LIN {X 0,Y 573.325,Z 84.689,A -85,B 0,C 180,E1 -2340.7,E2 -2340.7} C_VEL
LIN {X 0,Y 573.297,Z 84.693,A -85,B 0,C 180,E1 -2342.808,E2 -2342.808} C_VEL
LIN {X 0,Y 573.291,Z 84.697,A -85,B 0,C 180,E1 -2345.626,E2 -2345.626} C_VEL
LIN {X 0,Y 573.254,Z 84.699,A -85,B 0,C 180,E1 -2348.457,E2 -2348.457} C_VEL
LIN {X 0,Y 573.274,Z 84.699,A -85,B 0,C 180,E1 -2351.309,E2 -2351.309} C_VEL
LIN {X 0,Y 573.262,Z 84.697,A -85,B 0,C 180,E1 -2354.414,E2 -2354.414} C_VEL
LIN {X 0,Y 573.247,Z 84.702,A -85,B 0,C 180,E1 -2357.109,E2 -2357.109} C_VEL
LIN {X 0,Y 573.233,Z 84.701,A -85,B 0,C 180,E1 -2360.074,E2 -2360.074} C_VEL
LIN {X 0,Y 573.225,Z 84.702,A -85,B 0,C 180,E1 -2362.335,E2 -2362.335} C_VEL
LIN {X 0,Y 573.21,Z 84.704,A -85,B 0,C 180,E1 -2364.357,E2 -2364.357} C_VEL
LIN {X 0,Y 572.573,Z 84.79,A -85,B 0,C 180,E1 -2364.944,E2 -2364.944} C_VEL
LIN {X 0,Y 569.748,Z 85.144,A -85,B 0,C 180,E1 -2365.895,E2 -2365.895} C_VEL
LIN {X 0,Y 567.335,Z 85.445,A -85,B 0,C 180,E1 -2366.661,E2 -2366.661} C_VEL
LIN {X 0,Y 566.283,Z 85.573,A -85,B 0,C 180,E1 -2367.252,E2 -2367.252} C_VEL
LIN {X 0,Y 566.19,Z 85.582,A -85,B 0,C 180,E1 -2367.453,E2 -2367.453} C_VEL
LIN {X 0,Y 566.185,Z 85.576,A -85,B 0,C 180,E1 -2369.766,E2 -2369.766} C_VEL
LIN {X 0,Y 566.19,Z 85.581,A -85,B 0,C 180,E1 -2372.426,E2 -2372.426} C_VEL
LIN {X 0,Y 566.167,Z 85.588,A -85,B 0,C 180,E1 -2374.986,E2 -2374.986} C_VEL
LIN {X 0,Y 566.179,Z 85.579,A -85,B 0,C 180,E1 -2377.458,E2 -2377.458} C_VEL
LIN {X 0,Y 566.188,Z 85.583,A -85,B 0,C 180,E1 -2380.196,E2 -2380.196} C_VEL
LIN {X 0,Y 566.182,Z 85.582,A -85,B 0,C 180,E1 -2383.051,E2 -2383.051} C_VEL
LIN {X 0,Y 566.171,Z 85.585,A -85,B 0,C 180,E1 -2386.046,E2 -2386.046} C_VEL
LIN {X 0,Y 566.179,Z 85.583,A -85,B 0,C 180,E1 -2389.212,E2 -2389.212} C_VEL
LIN {X 0,Y 566.178,Z 85.589,A -85,B 0,C 180,E1 -2392.087,E2 -2392.087} C_VEL
LIN {X 0,Y 566.191,Z 85.725,A -85,B 0,C 180,E1 -2392.454,E2 -2392.454} C_VEL
LIN {X 0,Y 566.912,Z 90.584,A -85,B 0,C 180,E1 -2393.261,E2 -2393.261} C_VEL
LIN {X 0,Y 566.616,Z 108.38,A -85,B 0,C 180,E1 -2396.071,E2 -2396.071} C_VEL
LIN {X 0,Y 566.568,Z 114.772,A -85,B 0,C 180,E1 -2397.07,E2 -2397.07} C_VEL
LIN {X 0,Y 567.79,Z 122.54,A -85,B 0,C 180,E1 -2397.221,E2 -2397.221} C_VEL
LIN {X 0,Y 567.456,Z 251.252,A -85,B 0,C 180,E1 -2398.889,E2 -2398.889} C_VEL
LIN {X 0,Y 567.291,Z 265.503,A -85,B 0,C 180,E1 -2399.215,E2 -2399.215} C_VEL
LIN {X 0,Y 567.168,Z 279.065,A -85,B 0,C 180,E1 -2399.671,E2 -2399.671} C_VEL
LIN {X 0,Y 566.965,Z 292.537,A -85,B 0,C 180,E1 -2400.274,E2 -2400.274} C_VEL
LIN {X 0,Y 566.763,Z 304.844,A -85,B 0,C 180,E1 -2400.976,E2 -2400.976} C_VEL
LIN {X 0,Y 566.577,Z 316.448,A -85,B 0,C 180,E1 -2401.791,E2 -2401.791} C_VEL
LIN {X 0,Y 566.434,Z 326.814,A -85,B 0,C 180,E1 -2402.672,E2 -2402.672} C_VEL
LIN {X 0,Y 566.277,Z 336.543,A -85,B 0,C 180,E1 -2403.66,E2 -2403.66} C_VEL
LIN {X 0,Y 566.136,Z 346.301,A -85,B 0,C 180,E1 -2404.857,E2 -2404.857} C_VEL
LIN {X 0,Y 566.039,Z 353.975,A -85,B 0,C 180,E1 -2406.006,E2 -2406.006} C_VEL
LIN {X 0,Y 565.976,Z 359.753,A -85,B 0,C 180,E1 -2407.05,E2 -2407.05} C_VEL
LIN {X 0,Y 565.952,Z 365.875,A -85,B 0,C 180,E1 -2408.421,E2 -2408.421} C_VEL
LIN {X 0,Y 565.893,Z 370.084,A -85,B 0,C 180,E1 -2409.65,E2 -2409.65} C_VEL
LIN {X 0,Y 565.895,Z 372.821,A -85,B 0,C 180,E1 -2410.698,E2 -2410.698} C_VEL
LIN {X 0,Y 565.829,Z 375.002,A -85,B 0,C 180,E1 -2411.909,E2 -2411.909} C_VEL
LIN {X 0,Y 565.849,Z 376.362,A -85,B 0,C 180,E1 -2413.4,E2 -2413.4} C_VEL
LIN {X 0,Y 565.844,Z 376.254,A -85,B 0,C 180,E1 -2414.88,E2 -2414.88} C_VEL
LIN {X 0,Y 565.917,Z 375.67,A -85,B 0,C 180,E1 -2415.618,E2 -2415.618} C_VEL
LIN {X 0,Y 565.859,Z 373.452,A -85,B 0,C 180,E1 -2417.081,E2 -2417.081} C_VEL
LIN {X 0,Y 565.91,Z 369.79,A -85,B 0,C 180,E1 -2418.538,E2 -2418.538} C_VEL
LIN {X 0,Y 565.919,Z 366.053,A -85,B 0,C 180,E1 -2419.625,E2 -2419.625} C_VEL
LIN {X 0,Y 565.944,Z 361.413,A -85,B 0,C 180,E1 -2420.709,E2 -2420.709} C_VEL
LIN {X 0,Y 566.021,Z 354.686,A -85,B 0,C 180,E1 -2421.969,E2 -2421.969} C_VEL
LIN {X 0,Y 566.131,Z 346.236,A -85,B 0,C 180,E1 -2423.242,E2 -2423.242} C_VEL
LIN {X 0,Y 566.262,Z 337.713,A -85,B 0,C 180,E1 -2424.301,E2 -2424.301} C_VEL
LIN {X 0,Y 566.408,Z 327.309,A -85,B 0,C 180,E1 -2425.373,E2 -2425.373} C_VEL
LIN {X 0,Y 566.578,Z 315.73,A -85,B 0,C 180,E1 -2426.354,E2 -2426.354} C_VEL
LIN {X 0,Y 566.74,Z 304.194,A -85,B 0,C 180,E1 -2427.156,E2 -2427.156} C_VEL
LIN {X 0,Y 566.982,Z 291.521,A -85,B 0,C 180,E1 -2427.868,E2 -2427.868} C_VEL
LIN {X 0,Y 567.18,Z 278.421,A -85,B 0,C 180,E1 -2428.446,E2 -2428.446} C_VEL
LIN {X 0,Y 567.309,Z 264.238,A -85,B 0,C 180,E1 -2428.912,E2 -2428.912} C_VEL
LIN {X 0,Y 567.408,Z 250.022,A -85,B 0,C 180,E1 -2429.223,E2 -2429.223} C_VEL
LIN {X 0,Y 567.634,Z 120.855,A -85,B 0,C 180,E1 -2430.896,E2 -2430.896} C_VEL
LIN {X 0,Y 566.54,Z 114.763,A -85,B 0,C 180,E1 -2431.021,E2 -2431.021} C_VEL
LIN {X 0,Y 566.822,Z 95.22,A -85,B 0,C 180,E1 -2434.087,E2 -2434.087} C_VEL
LIN {X 0,Y 566.763,Z 88.525,A -85,B 0,C 180,E1 -2435.157,E2 -2435.157} C_VEL
LIN {X 0,Y 566.246,Z 85.58,A -85,B 0,C 180,E1 -2435.653,E2 -2435.653} C_VEL
LIN {X 0,Y 566.23,Z 85.582,A -85,B 0,C 180,E1 -2437.846,E2 -2437.846} C_VEL
LIN {X 0,Y 566.226,Z 85.575,A -85,B 0,C 180,E1 -2440.729,E2 -2440.729} C_VEL
LIN {X 0,Y 566.198,Z 85.587,A -85,B 0,C 180,E1 -2443.64,E2 -2443.64} C_VEL
LIN {X 0,Y 566.208,Z 85.575,A -85,B 0,C 180,E1 -2446.587,E2 -2446.587} C_VEL
LIN {X 0,Y 566.181,Z 85.588,A -85,B 0,C 180,E1 -2449.58,E2 -2449.58} C_VEL
LIN {X 0,Y 566.205,Z 85.576,A -85,B 0,C 180,E1 -2452.629,E2 -2452.629} C_VEL
LIN {X 0,Y 566.198,Z 85.58,A -85,B 0,C 180,E1 -2455.748,E2 -2455.748} C_VEL
LIN {X 0,Y 566.208,Z 85.575,A -85,B 0,C 180,E1 -2458.212,E2 -2458.212} C_VEL
LIN {X 0,Y 566.179,Z 85.587,A -85,B 0,C 180,E1 -2461.082,E2 -2461.082} C_VEL
LIN {X 0,Y 566.199,Z 85.578,A -85,B 0,C 180,E1 -2463.739,E2 -2463.739} C_VEL
LIN {X 0,Y 566.195,Z 85.58,A -85,B 0,C 180,E1 -2466.569,E2 -2466.569} C_VEL
LIN {X 0,Y 566.241,Z 85.572,A -85,B 0,C 180,E1 -2469.695,E2 -2469.695} C_VEL
LIN {X 0,Y 566.196,Z 85.577,A -85,B 0,C 180,E1 -2472.087,E2 -2472.087} C_VEL
LIN {X 0,Y 566.191,Z 85.583,A -85,B 0,C 180,E1 -2475.032,E2 -2475.032} C_VEL
LIN {X 0,Y 566.202,Z 85.578,A -85,B 0,C 180,E1 -2478.136,E2 -2478.136} C_VEL
LIN {X 0,Y 566.199,Z 85.584,A -85,B 0,C 180,E1 -2480.73,E2 -2480.73} C_VEL
LIN {X 0,Y 566.202,Z 85.577,A -85,B 0,C 180,E1 -2483.784,E2 -2483.784} C_VEL
LIN {X 0,Y 566.204,Z 85.583,A -85,B 0,C 180,E1 -2486.265,E2 -2486.265} C_VEL
LIN {X 0,Y 566.181,Z 85.58,A -85,B 0,C 180,E1 -2488.923,E2 -2488.923} C_VEL
LIN {X 0,Y 566.204,Z 85.579,A -85,B 0,C 180,E1 -2491.795,E2 -2491.795} C_VEL
LIN {X 0,Y 566.208,Z 85.583,A -85,B 0,C 180,E1 -2494.254,E2 -2494.254} C_VEL
LIN {X 0,Y 566.225,Z 85.575,A -85,B 0,C 180,E1 -2496.703,E2 -2496.703} C_VEL
LIN {X 0,Y 566.206,Z 85.58,A -85,B 0,C 180,E1 -2499.666,E2 -2499.666} C_VEL
LIN {X 0,Y 566.189,Z 85.578,A -85,B 0,C 180,E1 -2502.671,E2 -2502.671} C_VEL
LIN {X 0,Y 566.218,Z 85.581,A -85,B 0,C 180,E1 -2505.629,E2 -2505.629} C_VEL
LIN {X 0,Y 566.26,Z 85.569,A -85,B 0,C 180,E1 -2508.656,E2 -2508.656} C_VEL
LIN {X 0,Y 566.238,Z 85.578,A -85,B 0,C 180,E1 -2511.437,E2 -2511.437} C_VEL
LIN {X 0,Y 566.253,Z 85.57,A -85,B 0,C 180,E1 -2514.304,E2 -2514.304} C_VEL
LIN {X 0,Y 566.269,Z 85.571,A -85,B 0,C 180,E1 -2517.869,E2 -2517.869} C_VEL
LIN {X 0,Y 566.3,Z 85.565,A -85,B 0,C 180,E1 -2520.713,E2 -2520.713} C_VEL
LIN {X 0,Y 566.27,Z 85.571,A -85,B 0,C 180,E1 -2522.848,E2 -2522.848} C_VEL
LIN {X 0,Y 566.253,Z 85.572,A -85,B 0,C 180,E1 -2525.701,E2 -2525.701} C_VEL
LIN {X 0,Y 566.227,Z 85.575,A -85,B 0,C 180,E1 -2528.568,E2 -2528.568} C_VEL
LIN {X 0,Y 566.235,Z 85.575,A -85,B 0,C 180,E1 -2531.456,E2 -2531.456} C_VEL
LIN {X 0,Y 566.228,Z 85.577,A -85,B 0,C 180,E1 -2534.509,E2 -2534.509} C_VEL
LIN {X 0,Y 566.194,Z 85.579,A -85,B 0,C 180,E1 -2537.334,E2 -2537.334} C_VEL
LIN {X 0,Y 566.209,Z 85.579,A -85,B 0,C 180,E1 -2540.339,E2 -2540.339} C_VEL
LIN {X 0,Y 566.185,Z 85.579,A -85,B 0,C 180,E1 -2543.406,E2 -2543.406} C_VEL
LIN {X 0,Y 566.221,Z 85.574,A -85,B 0,C 180,E1 -2545.75,E2 -2545.75} C_VEL
LIN {X 0,Y 566.203,Z 85.581,A -85,B 0,C 180,E1 -2548.205,E2 -2548.205} C_VEL
LIN {X 0,Y 566.187,Z 85.579,A -85,B 0,C 180,E1 -2551.078,E2 -2551.078} C_VEL
LIN {X 0,Y 566.208,Z 85.577,A -85,B 0,C 180,E1 -2553.736,E2 -2553.736} C_VEL
LIN {X 0,Y 566.208,Z 85.579,A -85,B 0,C 180,E1 -2556.571,E2 -2556.571} C_VEL
LIN {X 0,Y 566.213,Z 85.578,A -85,B 0,C 180,E1 -2559.687,E2 -2559.687} C_VEL
LIN {X 0,Y 566.212,Z 85.584,A -85,B 0,C 180,E1 -2562.089,E2 -2562.089} C_VEL
LIN {X 0,Y 566.172,Z 85.58,A -85,B 0,C 180,E1 -2565.037,E2 -2565.037} C_VEL
LIN {X 0,Y 566.211,Z 85.58,A -85,B 0,C 180,E1 -2568.138,E2 -2568.138} C_VEL
LIN {X 0,Y 566.213,Z 85.575,A -85,B 0,C 180,E1 -2570.728,E2 -2570.728} C_VEL
LIN {X 0,Y 566.183,Z 85.586,A -85,B 0,C 180,E1 -2573.79,E2 -2573.79} C_VEL
LIN {X 0,Y 566.211,Z 85.576,A -85,B 0,C 180,E1 -2576.267,E2 -2576.267} C_VEL
LIN {X 0,Y 566.187,Z 85.581,A -85,B 0,C 180,E1 -2578.926,E2 -2578.926} C_VEL
LIN {X 0,Y 566.212,Z 85.58,A -85,B 0,C 180,E1 -2581.859,E2 -2581.859} C_VEL
LIN {X 0,Y 566.208,Z 85.579,A -85,B 0,C 180,E1 -2584.252,E2 -2584.252} C_VEL
LIN {X 0,Y 566.246,Z 85.676,A -85,B 0,C 180,E1 -2585.286,E2 -2585.286} C_VEL
LIN {X 0,Y 567.327,Z 92.177,A -85,B 0,C 180,E1 -2586.222,E2 -2586.222} C_VEL
LIN {X 0,Y 567.075,Z 112.447,A -85,B 0,C 180,E1 -2588.937,E2 -2588.937} C_VEL
LIN {X 0,Y 566.776,Z 135.267,A -85,B 0,C 180,E1 -2591.942,E2 -2591.942} C_VEL
LIN {X 0,Y 566.668,Z 143.53,A -85,B 0,C 180,E1 -2593.019,E2 -2593.019} C_VEL
LIN {X 0,Y 567.795,Z 150.908,A -85,B 0,C 180,E1 -2593.156,E2 -2593.156} C_VEL
LIN {X 0,Y 567.434,Z 281.941,A -85,B 0,C 180,E1 -2594.856,E2 -2594.856} C_VEL
LIN {X 0,Y 567.269,Z 296.626,A -85,B 0,C 180,E1 -2595.203,E2 -2595.203} C_VEL
LIN {X 0,Y 567.1,Z 310.862,A -85,B 0,C 180,E1 -2595.696,E2 -2595.696} C_VEL
LIN {X 0,Y 566.963,Z 323.66,A -85,B 0,C 180,E1 -2596.287,E2 -2596.287} C_VEL
LIN {X 0,Y 566.786,Z 336.117,A -85,B 0,C 180,E1 -2597.013,E2 -2597.013} C_VEL
LIN {X 0,Y 566.577,Z 347.497,A -85,B 0,C 180,E1 -2597.828,E2 -2597.828} C_VEL
LIN {X 0,Y 566.411,Z 358.022,A -85,B 0,C 180,E1 -2598.738,E2 -2598.738} C_VEL
LIN {X 0,Y 566.247,Z 368.343,A -85,B 0,C 180,E1 -2599.814,E2 -2599.814} C_VEL
LIN {X 0,Y 566.152,Z 376.919,A -85,B 0,C 180,E1 -2600.894,E2 -2600.894} C_VEL
LIN {X 0,Y 566.06,Z 385.123,A -85,B 0,C 180,E1 -2602.152,E2 -2602.152} C_VEL
LIN {X 0,Y 565.967,Z 391.807,A -85,B 0,C 180,E1 -2603.423,E2 -2603.423} C_VEL
LIN {X 0,Y 565.928,Z 396.964,A -85,B 0,C 180,E1 -2604.657,E2 -2604.657} C_VEL
LIN {X 0,Y 565.957,Z 400.447,A -85,B 0,C 180,E1 -2605.728,E2 -2605.728} C_VEL
LIN {X 0,Y 565.874,Z 403.834,A -85,B 0,C 180,E1 -2607.153,E2 -2607.153} C_VEL
LIN {X 0,Y 565.841,Z 405.835,A -85,B 0,C 180,E1 -2608.578,E2 -2608.578} C_VEL
LIN {X 0,Y 565.837,Z 406.5,A -85,B 0,C 180,E1 -2610.001,E2 -2610.001} C_VEL
LIN {X 0,Y 565.841,Z 405.834,A -85,B 0,C 180,E1 -2611.424,E2 -2611.424} C_VEL
LIN {X 0,Y 565.874,Z 403.833,A -85,B 0,C 180,E1 -2612.849,E2 -2612.849} C_VEL
LIN {X 0,Y 565.957,Z 400.443,A -85,B 0,C 180,E1 -2614.274,E2 -2614.274} C_VEL
LIN {X 0,Y 565.986,Z 395.564,A -85,B 0,C 180,E1 -2615.702,E2 -2615.702} C_VEL
LIN {X 0,Y 565.998,Z 391.039,A -85,B 0,C 180,E1 -2616.74,E2 -2616.74} C_VEL
LIN {X 0,Y 566.049,Z 384.03,A -85,B 0,C 180,E1 -2618.03,E2 -2618.03} C_VEL
LIN {X 0,Y 566.178,Z 375.549,A -85,B 0,C 180,E1 -2619.287,E2 -2619.287} C_VEL
LIN {X 0,Y 566.295,Z 366.698,A -85,B 0,C 180,E1 -2620.368,E2 -2620.368} C_VEL
LIN {X 0,Y 566.471,Z 355.976,A -85,B 0,C 180,E1 -2621.451,E2 -2621.451} C_VEL
LIN {X 0,Y 566.632,Z 345.123,A -85,B 0,C 180,E1 -2622.355,E2 -2622.355} C_VEL
LIN {X 0,Y 566.801,Z 333.237,A -85,B 0,C 180,E1 -2623.171,E2 -2623.171} C_VEL
LIN {X 0,Y 567.027,Z 320.076,A -85,B 0,C 180,E1 -2623.896,E2 -2623.896} C_VEL
LIN {X 0,Y 567.236,Z 307.029,A -85,B 0,C 180,E1 -2624.453,E2 -2624.453} C_VEL
LIN {X 0,Y 567.329,Z 293.201,A -85,B 0,C 180,E1 -2624.893,E2 -2624.893} C_VEL
LIN {X 0,Y 567.433,Z 279.065,A -85,B 0,C 180,E1 -2625.192,E2 -2625.192} C_VEL
LIN {X 0,Y 567.737,Z 149.617,A -85,B 0,C 180,E1 -2626.863,E2 -2626.863} C_VEL
LIN {X 0,Y 566.67,Z 143.509,A -85,B 0,C 180,E1 -2626.983,E2 -2626.983} C_VEL
LIN {X 0,Y 566.939,Z 122.534,A -85,B 0,C 180,E1 -2629.725,E2 -2629.725} C_VEL
LIN {X 0,Y 567.157,Z 100.948,A -85,B 0,C 180,E1 -2632.591,E2 -2632.591} C_VEL
LIN {X 0,Y 567.257,Z 90.849,A -85,B 0,C 180,E1 -2633.956,E2 -2633.956} C_VEL
LIN {X 0,Y 566.197,Z 85.587,A -85,B 0,C 180,E1 -2634.743,E2 -2634.743} C_VEL
LIN {X 0,Y 566.202,Z 85.578,A -85,B 0,C 180,E1 -2637.341,E2 -2637.341} C_VEL
LIN {X 0,Y 566.205,Z 85.579,A -85,B 0,C 180,E1 -2639.77,E2 -2639.77} C_VEL
LIN {X 0,Y 566.212,Z 85.584,A -85,B 0,C 180,E1 -2642.43,E2 -2642.43} C_VEL
LIN {X 0,Y 566.187,Z 85.58,A -85,B 0,C 180,E1 -2644.989,E2 -2644.989} C_VEL
LIN {X 0,Y 566.203,Z 85.577,A -85,B 0,C 180,E1 -2647.461,E2 -2647.461} C_VEL
LIN {X 0,Y 566.217,Z 85.581,A -85,B 0,C 180,E1 -2650.199,E2 -2650.199} C_VEL
LIN {X 0,Y 566.198,Z 85.577,A -85,B 0,C 180,E1 -2653.056,E2 -2653.056} C_VEL
LIN {X 0,Y 566.205,Z 85.583,A -85,B 0,C 180,E1 -2656.049,E2 -2656.049} C_VEL
LIN {X 0,Y 566.215,Z 85.574,A -85,B 0,C 180,E1 -2659.214,E2 -2659.214} C_VEL
LIN {X 0,Y 566.192,Z 85.587,A -85,B 0,C 180,E1 -2661.636,E2 -2661.636} C_VEL
LIN {X 0,Y 566.161,Z 85.582,A -85,B 0,C 180,E1 -2664.306,E2 -2664.306} C_VEL
LIN {X 0,Y 566.211,Z 85.577,A -85,B 0,C 180,E1 -2666.896,E2 -2666.896} C_VEL
LIN {X 0,Y 566.183,Z 85.587,A -85,B 0,C 180,E1 -2669.406,E2 -2669.406} C_VEL
LIN {X 0,Y 566.2,Z 85.577,A -85,B 0,C 180,E1 -2671.855,E2 -2671.855} C_VEL
LIN {X 0,Y 566.25,Z 85.579,A -85,B 0,C 180,E1 -2675.038,E2 -2675.038} C_VEL
LIN {X 0,Y 566.199,Z 85.577,A -85,B 0,C 180,E1 -2678.136,E2 -2678.136} C_VEL
LIN {X 0,Y 566.243,Z 85.575,A -85,B 0,C 180,E1 -2680.613,E2 -2680.613} C_VEL
LIN {X 0,Y 566.212,Z 85.575,A -85,B 0,C 180,E1 -2683.41,E2 -2683.41} C_VEL
LIN {X 0,Y 566.198,Z 85.582,A -85,B 0,C 180,E1 -2686.357,E2 -2686.357} C_VEL
LIN {X 0,Y 566.246,Z 85.579,A -85,B 0,C 180,E1 -2688.674,E2 -2688.674} C_VEL
LIN {X 0,Y 566.211,Z 85.575,A -85,B 0,C 180,E1 -2691.432,E2 -2691.432} C_VEL
LIN {X 0,Y 566.251,Z 85.578,A -85,B 0,C 180,E1 -2694.299,E2 -2694.299} C_VEL
LIN {X 0,Y 566.285,Z 85.569,A -85,B 0,C 180,E1 -2697.864,E2 -2697.864} C_VEL
LIN {X 0,Y 566.297,Z 85.565,A -85,B 0,C 180,E1 -2700.709,E2 -2700.709} C_VEL
LIN {X 0,Y 566.265,Z 85.569,A -85,B 0,C 180,E1 -2702.843,E2 -2702.843} C_VEL
LIN {X 0,Y 566.258,Z 85.574,A -85,B 0,C 180,E1 -2705.696,E2 -2705.696} C_VEL
LIN {X 0,Y 566.206,Z 85.576,A -85,B 0,C 180,E1 -2708.563,E2 -2708.563} C_VEL
LIN {X 0,Y 566.244,Z 85.577,A -85,B 0,C 180,E1 -2711.451,E2 -2711.451} C_VEL
LIN {X 0,Y 566.218,Z 85.575,A -85,B 0,C 180,E1 -2714.497,E2 -2714.497} C_VEL
LIN {X 0,Y 566.19,Z 85.584,A -85,B 0,C 180,E1 -2717.329,E2 -2717.329} C_VEL
LIN {X 0,Y 566.2,Z 85.576,A -85,B 0,C 180,E1 -2720.334,E2 -2720.334} C_VEL
LIN {X 0,Y 566.161,Z 85.59,A -85,B 0,C 180,E1 -2723.277,E2 -2723.277} C_VEL
LIN {X 0,Y 566.195,Z 85.578,A -85,B 0,C 180,E1 -2725.746,E2 -2725.746} C_VEL
LIN {X 0,Y 566.19,Z 85.582,A -85,B 0,C 180,E1 -2727.453,E2 -2727.453} C_VEL
LIN {X 0,Y 565.501,Z 85.666,A -85,B 0,C 180,E1 -2728.046,E2 -2728.046} C_VEL
LIN {X 0,Y 562.635,Z 86.027,A -85,B 0,C 180,E1 -2729.01,E2 -2729.01} C_VEL
LIN {X 0,Y 560.23,Z 86.321,A -85,B 0,C 180,E1 -2729.786,E2 -2729.786} C_VEL
LIN {X 0,Y 559.204,Z 86.447,A -85,B 0,C 180,E1 -2730.384,E2 -2730.384} C_VEL
LIN {X 0,Y 559.123,Z 86.459,A -85,B 0,C 180,E1 -2730.587,E2 -2730.587} C_VEL
LIN {X 0,Y 559.139,Z 86.463,A -85,B 0,C 180,E1 -2732.712,E2 -2732.712} C_VEL
LIN {X 0,Y 559.114,Z 86.462,A -85,B 0,C 180,E1 -2735.321,E2 -2735.321} C_VEL
LIN {X 0,Y 559.113,Z 86.459,A -85,B 0,C 180,E1 -2738.015,E2 -2738.015} C_VEL
LIN {X 0,Y 559.139,Z 86.462,A -85,B 0,C 180,E1 -2740.809,E2 -2740.809} C_VEL
LIN {X 0,Y 559.126,Z 86.46,A -85,B 0,C 180,E1 -2743.193,E2 -2743.193} C_VEL
LIN {X 0,Y 559.114,Z 86.468,A -85,B 0,C 180,E1 -2746.262,E2 -2746.262} C_VEL
LIN {X 0,Y 559.13,Z 86.462,A -85,B 0,C 180,E1 -2749.184,E2 -2749.184} C_VEL
LIN {X 0,Y 559.176,Z 86.575,A -85,B 0,C 180,E1 -2752.282,E2 -2752.282} C_VEL
LIN {X 0,Y 559.989,Z 92.284,A -85,B 0,C 180,E1 -2753.24,E2 -2753.24} C_VEL
LIN {X 0,Y 559.67,Z 109.35,A -85,B 0,C 180,E1 -2755.967,E2 -2755.967} C_VEL
LIN {X 0,Y 559.617,Z 114.96,A -85,B 0,C 180,E1 -2756.852,E2 -2756.852} C_VEL
LIN {X 0,Y 561,Z 122.414,A -85,B 0,C 180,E1 -2757.007,E2 -2757.007} C_VEL
LIN {X 0,Y 560.611,Z 251.638,A -85,B 0,C 180,E1 -2758.704,E2 -2758.704} C_VEL
LIN {X 0,Y 560.421,Z 265.852,A -85,B 0,C 180,E1 -2759.036,E2 -2759.036} C_VEL
LIN {X 0,Y 560.293,Z 279.873,A -85,B 0,C 180,E1 -2759.52,E2 -2759.52} C_VEL
LIN {X 0,Y 560.063,Z 292.156,A -85,B 0,C 180,E1 -2760.078,E2 -2760.078} C_VEL
LIN {X 0,Y 559.837,Z 304.514,A -85,B 0,C 180,E1 -2760.788,E2 -2760.788} C_VEL
LIN {X 0,Y 559.601,Z 317.408,A -85,B 0,C 180,E1 -2761.712,E2 -2761.712} C_VEL
LIN {X 0,Y 559.402,Z 328.703,A -85,B 0,C 180,E1 -2762.705,E2 -2762.705} C_VEL
LIN {X 0,Y 559.223,Z 338.11,A -85,B 0,C 180,E1 -2763.703,E2 -2763.703} C_VEL
LIN {X 0,Y 559.082,Z 346.929,A -85,B 0,C 180,E1 -2764.825,E2 -2764.825} C_VEL
LIN {X 0,Y 558.973,Z 355.021,A -85,B 0,C 180,E1 -2766.078,E2 -2766.078} C_VEL
LIN {X 0,Y 558.884,Z 362.079,A -85,B 0,C 180,E1 -2767.446,E2 -2767.446} C_VEL
LIN {X 0,Y 558.85,Z 366.88,A -85,B 0,C 180,E1 -2768.61,E2 -2768.61} C_VEL
LIN {X 0,Y 558.821,Z 370.587,A -85,B 0,C 180,E1 -2769.765,E2 -2769.765} C_VEL
LIN {X 0,Y 558.786,Z 373.335,A -85,B 0,C 180,E1 -2770.912,E2 -2770.912} C_VEL
LIN {X 0,Y 558.74,Z 375.645,A -85,B 0,C 180,E1 -2772.429,E2 -2772.429} C_VEL
LIN {X 0,Y 558.741,Z 376.482,A -85,B 0,C 180,E1 -2773.934,E2 -2773.934} C_VEL
LIN {X 0,Y 558.782,Z 375.89,A -85,B 0,C 180,E1 -2775.43,E2 -2775.43} C_VEL
LIN {X 0,Y 558.758,Z 373.862,A -85,B 0,C 180,E1 -2776.914,E2 -2776.914} C_VEL
LIN {X 0,Y 558.82,Z 370.391,A -85,B 0,C 180,E1 -2778.39,E2 -2778.39} C_VEL
LIN {X 0,Y 558.847,Z 365.414,A -85,B 0,C 180,E1 -2779.859,E2 -2779.859} C_VEL
LIN {X 0,Y 558.914,Z 358.797,A -85,B 0,C 180,E1 -2781.32,E2 -2781.32} C_VEL
LIN {X 0,Y 559.023,Z 351.462,A -85,B 0,C 180,E1 -2782.595,E2 -2782.595} C_VEL
LIN {X 0,Y 559.124,Z 343.814,A -85,B 0,C 180,E1 -2783.685,E2 -2783.685} C_VEL
LIN {X 0,Y 559.278,Z 334.677,A -85,B 0,C 180,E1 -2784.772,E2 -2784.772} C_VEL
LIN {X 0,Y 559.427,Z 325.61,A -85,B 0,C 180,E1 -2785.676,E2 -2785.676} C_VEL
LIN {X 0,Y 559.656,Z 313.679,A -85,B 0,C 180,E1 -2786.669,E2 -2786.669} C_VEL
LIN {X 0,Y 559.856,Z 301.71,A -85,B 0,C 180,E1 -2787.481,E2 -2787.481} C_VEL
LIN {X 0,Y 560.137,Z 288.323,A -85,B 0,C 180,E1 -2788.201,E2 -2788.201} C_VEL
LIN {X 0,Y 560.333,Z 275.423,A -85,B 0,C 180,E1 -2788.741,E2 -2788.741} C_VEL
LIN {X 0,Y 560.449,Z 261.6,A -85,B 0,C 180,E1 -2789.168,E2 -2789.168} C_VEL
LIN {X 0,Y 560.556,Z 247.05,A -85,B 0,C 180,E1 -2789.46,E2 -2789.46} C_VEL
LIN {X 0,Y 560.931,Z 122.222,A -85,B 0,C 180,E1 -2791.087,E2 -2791.087} C_VEL
LIN {X 0,Y 559.599,Z 114.957,A -85,B 0,C 180,E1 -2791.236,E2 -2791.236} C_VEL
LIN {X 0,Y 559.912,Z 95.543,A -85,B 0,C 180,E1 -2794.318,E2 -2794.318} C_VEL
LIN {X 0,Y 559.83,Z 89.958,A -85,B 0,C 180,E1 -2795.221,E2 -2795.221} C_VEL
LIN {X 0,Y 559.211,Z 86.457,A -85,B 0,C 180,E1 -2795.815,E2 -2795.815} C_VEL
LIN {X 0,Y 559.179,Z 86.453,A -85,B 0,C 180,E1 -2798.673,E2 -2798.673} C_VEL
LIN {X 0,Y 559.171,Z 86.46,A -85,B 0,C 180,E1 -2801.6,E2 -2801.6} C_VEL
LIN {X 0,Y 559.199,Z 86.448,A -85,B 0,C 180,E1 -2804.611,E2 -2804.611} C_VEL
LIN {X 0,Y 559.176,Z 86.46,A -85,B 0,C 180,E1 -2807.555,E2 -2807.555} C_VEL
LIN {X 0,Y 559.158,Z 86.454,A -85,B 0,C 180,E1 -2810.604,E2 -2810.604} C_VEL
LIN {X 0,Y 559.16,Z 86.458,A -85,B 0,C 180,E1 -2813.715,E2 -2813.715} C_VEL
LIN {X 0,Y 559.171,Z 86.452,A -85,B 0,C 180,E1 -2816.096,E2 -2816.096} C_VEL
LIN {X 0,Y 559.151,Z 86.455,A -85,B 0,C 180,E1 -2818.529,E2 -2818.529} C_VEL
LIN {X 0,Y 559.146,Z 86.463,A -85,B 0,C 180,E1 -2821.281,E2 -2821.281} C_VEL
LIN {X 0,Y 559.155,Z 86.454,A -85,B 0,C 180,E1 -2823.955,E2 -2823.955} C_VEL
LIN {X 0,Y 559.172,Z 86.454,A -85,B 0,C 180,E1 -2826.455,E2 -2826.455} C_VEL
LIN {X 0,Y 559.201,Z 86.448,A -85,B 0,C 180,E1 -2829.862,E2 -2829.862} C_VEL
LIN {X 0,Y 559.141,Z 86.464,A -85,B 0,C 180,E1 -2832.744,E2 -2832.744} C_VEL
LIN {X 0,Y 559.156,Z 86.454,A -85,B 0,C 180,E1 -2835.759,E2 -2835.759} C_VEL
LIN {X 0,Y 559.168,Z 86.457,A -85,B 0,C 180,E1 -2838.947,E2 -2838.947} C_VEL
LIN {X 0,Y 559.152,Z 86.456,A -85,B 0,C 180,E1 -2841.193,E2 -2841.193} C_VEL
LIN {X 0,Y 559.157,Z 86.455,A -85,B 0,C 180,E1 -2843.795,E2 -2843.795} C_VEL
LIN {X 0,Y 559.153,Z 86.463,A -85,B 0,C 180,E1 -2846.429,E2 -2846.429} C_VEL
LIN {X 0,Y 559.145,Z 86.456,A -85,B 0,C 180,E1 -2848.984,E2 -2848.984} C_VEL
LIN {X 0,Y 559.159,Z 86.455,A -85,B 0,C 180,E1 -2851.618,E2 -2851.618} C_VEL
LIN {X 0,Y 559.182,Z 86.456,A -85,B 0,C 180,E1 -2853.907,E2 -2853.907} C_VEL
LIN {X 0,Y 559.16,Z 86.453,A -85,B 0,C 180,E1 -2857.072,E2 -2857.072} C_VEL
LIN {X 0,Y 559.17,Z 86.454,A -85,B 0,C 180,E1 -2859.398,E2 -2859.398} C_VEL
LIN {X 0,Y 559.148,Z 86.457,A -85,B 0,C 180,E1 -2862.446,E2 -2862.446} C_VEL
LIN {X 0,Y 559.178,Z 86.455,A -85,B 0,C 180,E1 -2865.444,E2 -2865.444} C_VEL
LIN {X 0,Y 559.21,Z 86.447,A -85,B 0,C 180,E1 -2868.596,E2 -2868.596} C_VEL
LIN {X 0,Y 559.193,Z 86.454,A -85,B 0,C 180,E1 -2871.328,E2 -2871.328} C_VEL
LIN {X 0,Y 559.221,Z 86.446,A -85,B 0,C 180,E1 -2874.232,E2 -2874.232} C_VEL
LIN {X 0,Y 559.237,Z 86.448,A -85,B 0,C 180,E1 -2877.121,E2 -2877.121} C_VEL
LIN {X 0,Y 559.249,Z 86.443,A -85,B 0,C 180,E1 -2880.002,E2 -2880.002} C_VEL
LIN {X 0,Y 559.236,Z 86.448,A -85,B 0,C 180,E1 -2882.884,E2 -2882.884} C_VEL
LIN {X 0,Y 559.222,Z 86.447,A -85,B 0,C 180,E1 -2885.772,E2 -2885.772} C_VEL
LIN {X 0,Y 559.185,Z 86.454,A -85,B 0,C 180,E1 -2888.676,E2 -2888.676} C_VEL
LIN {X 0,Y 559.198,Z 86.45,A -85,B 0,C 180,E1 -2891.603,E2 -2891.603} C_VEL
LIN {X 0,Y 559.193,Z 86.454,A -85,B 0,C 180,E1 -2894.598,E2 -2894.598} C_VEL
LIN {X 0,Y 559.154,Z 86.455,A -85,B 0,C 180,E1 -2897.559,E2 -2897.559} C_VEL
LIN {X 0,Y 559.167,Z 86.452,A -85,B 0,C 180,E1 -2899.839,E2 -2899.839} C_VEL
LIN {X 0,Y 559.137,Z 86.459,A -85,B 0,C 180,E1 -2902.155,E2 -2902.155} C_VEL
LIN {X 0,Y 559.176,Z 86.453,A -85,B 0,C 180,E1 -2905.189,E2 -2905.189} C_VEL
LIN {X 0,Y 559.191,Z 86.45,A -85,B 0,C 180,E1 -2907.713,E2 -2907.713} C_VEL
LIN {X 0,Y 559.15,Z 86.46,A -85,B 0,C 180,E1 -2910.185,E2 -2910.185} C_VEL
LIN {X 0,Y 559.172,Z 86.456,A -85,B 0,C 180,E1 -2912.716,E2 -2912.716} C_VEL
LIN {X 0,Y 559.142,Z 86.456,A -85,B 0,C 180,E1 -2915.325,E2 -2915.325} C_VEL
LIN {X 0,Y 559.131,Z 86.464,A -85,B 0,C 180,E1 -2918.019,E2 -2918.019} C_VEL
LIN {X 0,Y 559.157,Z 86.454,A -85,B 0,C 180,E1 -2920.814,E2 -2920.814} C_VEL
LIN {X 0,Y 559.147,Z 86.455,A -85,B 0,C 180,E1 -2923.198,E2 -2923.198} C_VEL
LIN {X 0,Y 559.139,Z 86.46,A -85,B 0,C 180,E1 -2926.268,E2 -2926.268} C_VEL
LIN {X 0,Y 559.164,Z 86.453,A -85,B 0,C 180,E1 -2928.95,E2 -2928.95} C_VEL
LIN {X 0,Y 559.174,Z 86.453,A -85,B 0,C 180,E1 -2931.193,E2 -2931.193} C_VEL
LIN {X 0,Y 559.138,Z 86.464,A -85,B 0,C 180,E1 -2933.791,E2 -2933.791} C_VEL
LIN {X 0,Y 559.158,Z 86.454,A -85,B 0,C 180,E1 -2936.426,E2 -2936.426} C_VEL
LIN {X 0,Y 559.151,Z 86.458,A -85,B 0,C 180,E1 -2938.982,E2 -2938.982} C_VEL
LIN {X 0,Y 559.168,Z 86.461,A -85,B 0,C 180,E1 -2941.62,E2 -2941.62} C_VEL
LIN {X 0,Y 559.177,Z 86.457,A -85,B 0,C 180,E1 -2943.904,E2 -2943.904} C_VEL
LIN {X 0,Y 559.219,Z 86.62,A -85,B 0,C 180,E1 -2945.106,E2 -2945.106} C_VEL
LIN {X 0,Y 560.437,Z 93.88,A -85,B 0,C 180,E1 -2946.166,E2 -2946.166} C_VEL
LIN {X 0,Y 560.098,Z 115.132,A -85,B 0,C 180,E1 -2949.048,E2 -2949.048} C_VEL
LIN {X 0,Y 559.808,Z 136.525,A -85,B 0,C 180,E1 -2951.899,E2 -2951.899} C_VEL
LIN {X 0,Y 559.699,Z 143.409,A -85,B 0,C 180,E1 -2952.808,E2 -2952.808} C_VEL
LIN {X 0,Y 560.995,Z 150.933,A -85,B 0,C 180,E1 -2952.949,E2 -2952.949} C_VEL
LIN {X 0,Y 560.593,Z 281.834,A -85,B 0,C 180,E1 -2954.667,E2 -2954.667} C_VEL
LIN {X 0,Y 560.441,Z 296.394,A -85,B 0,C 180,E1 -2955.013,E2 -2955.013} C_VEL
LIN {X 0,Y 560.212,Z 310.822,A -85,B 0,C 180,E1 -2955.516,E2 -2955.516} C_VEL
LIN {X 0,Y 560.057,Z 323.657,A -85,B 0,C 180,E1 -2956.115,E2 -2956.115} C_VEL
LIN {X 0,Y 559.841,Z 336.114,A -85,B 0,C 180,E1 -2956.849,E2 -2956.849} C_VEL
LIN {X 0,Y 559.617,Z 347.494,A -85,B 0,C 180,E1 -2957.674,E2 -2957.674} C_VEL
LIN {X 0,Y 559.388,Z 358.77,A -85,B 0,C 180,E1 -2958.666,E2 -2958.666} C_VEL
LIN {X 0,Y 559.239,Z 368.343,A -85,B 0,C 180,E1 -2959.685,E2 -2959.685} C_VEL
LIN {X 0,Y 559.114,Z 376.918,A -85,B 0,C 180,E1 -2960.779,E2 -2960.779} C_VEL
LIN {X 0,Y 558.98,Z 385.124,A -85,B 0,C 180,E1 -2962.051,E2 -2962.051} C_VEL
LIN {X 0,Y 558.895,Z 392.17,A -85,B 0,C 180,E1 -2963.421,E2 -2963.421} C_VEL
LIN {X 0,Y 558.858,Z 396.964,A -85,B 0,C 180,E1 -2964.589,E2 -2964.589} C_VEL
LIN {X 0,Y 558.866,Z 400.447,A -85,B 0,C 180,E1 -2965.674,E2 -2965.674} C_VEL
LIN {X 0,Y 558.795,Z 403.834,A -85,B 0,C 180,E1 -2967.117,E2 -2967.117} C_VEL
LIN {X 0,Y 558.741,Z 405.835,A -85,B 0,C 180,E1 -2968.56,E2 -2968.56} C_VEL
LIN {X 0,Y 558.738,Z 406.5,A -85,B 0,C 180,E1 -2970.001,E2 -2970.001} C_VEL
LIN {X 0,Y 558.741,Z 405.834,A -85,B 0,C 180,E1 -2971.443,E2 -2971.443} C_VEL
LIN {X 0,Y 558.796,Z 403.833,A -85,B 0,C 180,E1 -2972.885,E2 -2972.885} C_VEL
LIN {X 0,Y 558.866,Z 400.444,A -85,B 0,C 180,E1 -2974.328,E2 -2974.328} C_VEL
LIN {X 0,Y 558.915,Z 395.564,A -85,B 0,C 180,E1 -2975.774,E2 -2975.774} C_VEL
LIN {X 0,Y 558.906,Z 390.859,A -85,B 0,C 180,E1 -2976.861,E2 -2976.861} C_VEL
LIN {X 0,Y 558.988,Z 384.029,A -85,B 0,C 180,E1 -2978.132,E2 -2978.132} C_VEL
LIN {X 0,Y 559.119,Z 375.549,A -85,B 0,C 180,E1 -2979.406,E2 -2979.406} C_VEL
LIN {X 0,Y 559.274,Z 366.698,A -85,B 0,C 180,E1 -2980.5,E2 -2980.5} C_VEL
LIN {X 0,Y 559.458,Z 355.975,A -85,B 0,C 180,E1 -2981.596,E2 -2981.596} C_VEL
LIN {X 0,Y 559.643,Z 345.12,A -85,B 0,C 180,E1 -2982.512,E2 -2982.512} C_VEL
LIN {X 0,Y 559.842,Z 333.234,A -85,B 0,C 180,E1 -2983.338,E2 -2983.338} C_VEL
LIN {X 0,Y 560.109,Z 320.065,A -85,B 0,C 180,E1 -2984.071,E2 -2984.071} C_VEL
LIN {X 0,Y 560.356,Z 307.216,A -85,B 0,C 180,E1 -2984.626,E2 -2984.626} C_VEL
LIN {X 0,Y 560.455,Z 293.854,A -85,B 0,C 180,E1 -2985.061,E2 -2985.061} C_VEL
LIN {X 0,Y 560.589,Z 280.443,A -85,B 0,C 180,E1 -2985.358,E2 -2985.358} C_VEL
LIN {X 0,Y 560.883,Z 150.235,A -85,B 0,C 180,E1 -2987.064,E2 -2987.064} C_VEL
LIN {X 0,Y 559.715,Z 143.373,A -85,B 0,C 180,E1 -2987.193,E2 -2987.193} C_VEL
LIN {X 0,Y 560.017,Z 120.78,A -85,B 0,C 180,E1 -2990.19,E2 -2990.19} C_VEL
LIN {X 0,Y 560.387,Z 97.933,A -85,B 0,C 180,E1 -2993.27,E2 -2993.27} C_VEL
LIN {X 0,Y 560.345,Z 92.235,A -85,B 0,C 180,E1 -2994.056,E2 -2994.056} C_VEL
LIN {X 0,Y 559.165,Z 86.462,A -85,B 0,C 180,E1 -2994.919,E2 -2994.919} C_VEL
LIN {X 0,Y 559.149,Z 86.457,A -85,B 0,C 180,E1 -2997.715,E2 -2997.715} C_VEL
LIN {X 0,Y 559.157,Z 86.461,A -85,B 0,C 180,E1 -3000.184,E2 -3000.184} C_VEL
LIN {X 0,Y 559.162,Z 86.46,A -85,B 0,C 180,E1 -3002.716,E2 -3002.716} C_VEL
LIN {X 0,Y 559.132,Z 86.458,A -85,B 0,C 180,E1 -3005.325,E2 -3005.325} C_VEL
LIN {X 0,Y 559.142,Z 86.462,A -85,B 0,C 180,E1 -3008.018,E2 -3008.018} C_VEL
LIN {X 0,Y 559.166,Z 86.453,A -85,B 0,C 180,E1 -3010.813,E2 -3010.813} C_VEL
LIN {X 0,Y 559.122,Z 86.465,A -85,B 0,C 180,E1 -3013.737,E2 -3013.737} C_VEL
LIN {X 0,Y 559.149,Z 86.459,A -85,B 0,C 180,E1 -3016.266,E2 -3016.266} C_VEL
LIN {X 0,Y 559.167,Z 86.451,A -85,B 0,C 180,E1 -3019.187,E2 -3019.187} C_VEL
LIN {X 0,Y 559.14,Z 86.459,A -85,B 0,C 180,E1 -3021.982,E2 -3021.982} C_VEL
LIN {X 0,Y 559.14,Z 86.457,A -85,B 0,C 180,E1 -3024.787,E2 -3024.787} C_VEL
LIN {X 0,Y 559.165,Z 86.462,A -85,B 0,C 180,E1 -3027.364,E2 -3027.364} C_VEL
LIN {X 0,Y 559.134,Z 86.457,A -85,B 0,C 180,E1 -3030.147,E2 -3030.147} C_VEL
LIN {X 0,Y 559.155,Z 86.462,A -85,B 0,C 180,E1 -3033.177,E2 -3033.177} C_VEL
LIN {X 0,Y 559.166,Z 86.455,A -85,B 0,C 180,E1 -3035.494,E2 -3035.494} C_VEL
LIN {X 0,Y 559.183,Z 86.455,A -85,B 0,C 180,E1 -3038.623,E2 -3038.623} C_VEL
LIN {X 0,Y 559.171,Z 86.461,A -85,B 0,C 180,E1 -3040.925,E2 -3040.925} C_VEL
LIN {X 0,Y 559.166,Z 86.452,A -85,B 0,C 180,E1 -3043.946,E2 -3043.946} C_VEL
LIN {X 0,Y 559.172,Z 86.455,A -85,B 0,C 180,E1 -3046.182,E2 -3046.182} C_VEL
LIN {X 0,Y 559.202,Z 86.45,A -85,B 0,C 180,E1 -3049.132,E2 -3049.132} C_VEL
LIN {X 0,Y 559.199,Z 86.452,A -85,B 0,C 180,E1 -3052.051,E2 -3052.051} C_VEL
LIN {X 0,Y 559.25,Z 86.444,A -85,B 0,C 180,E1 -3054.951,E2 -3054.951} C_VEL
LIN {X 0,Y 559.257,Z 86.444,A -85,B 0,C 180,E1 -3057.837,E2 -3057.837} C_VEL
LIN {X 0,Y 559.269,Z 86.44,A -85,B 0,C 180,E1 -3060.718,E2 -3060.718} C_VEL
LIN {X 0,Y 559.233,Z 86.445,A -85,B 0,C 180,E1 -3062.879,E2 -3062.879} C_VEL
LIN {X 0,Y 559.226,Z 86.451,A -85,B 0,C 180,E1 -3065.768,E2 -3065.768} C_VEL
LIN {X 0,Y 559.17,Z 86.452,A -85,B 0,C 180,E1 -3068.672,E2 -3068.672} C_VEL
LIN {X 0,Y 559.207,Z 86.456,A -85,B 0,C 180,E1 -3071.598,E2 -3071.598} C_VEL
LIN {X 0,Y 559.181,Z 86.451,A -85,B 0,C 180,E1 -3074.585,E2 -3074.585} C_VEL
LIN {X 0,Y 559.134,Z 86.465,A -85,B 0,C 180,E1 -3077.555,E2 -3077.555} C_VEL
LIN {X 0,Y 559.161,Z 86.456,A -85,B 0,C 180,E1 -3079.835,E2 -3079.835} C_VEL
LIN {X 0,Y 559.134,Z 86.457,A -85,B 0,C 180,E1 -3082.15,E2 -3082.15} C_VEL
LIN {X 0,Y 559.135,Z 86.466,A -85,B 0,C 180,E1 -3085.175,E2 -3085.175} C_VEL
LIN {X 0,Y 559.138,Z 86.458,A -85,B 0,C 180,E1 -3087.711,E2 -3087.711} C_VEL
LIN {X 0,Y 559.123,Z 86.459,A -85,B 0,C 180,E1 -3090.587,E2 -3090.587} C_VEL
LIN {X 0,Y 558.46,Z 86.548,A -85,B 0,C 180,E1 -3091.189,E2 -3091.189} C_VEL
LIN {X 0,Y 555.597,Z 86.903,A -85,B 0,C 180,E1 -3092.165,E2 -3092.165} C_VEL
LIN {X 0,Y 553.181,Z 87.205,A -85,B 0,C 180,E1 -3092.95,E2 -3092.95} C_VEL
LIN {X 0,Y 552.154,Z 87.326,A -85,B 0,C 180,E1 -3093.557,E2 -3093.557} C_VEL
LIN {X 0,Y 552.076,Z 87.334,A -85,B 0,C 180,E1 -3093.762,E2 -3093.762} C_VEL
LIN {X 0,Y 552.09,Z 87.342,A -85,B 0,C 180,E1 -3096.744,E2 -3096.744} C_VEL
LIN {X 0,Y 552.109,Z 87.333,A -85,B 0,C 180,E1 -3099.524,E2 -3099.524} C_VEL
LIN {X 0,Y 552.113,Z 87.34,A -85,B 0,C 180,E1 -3102.422,E2 -3102.422} C_VEL
LIN {X 0,Y 552.071,Z 87.337,A -85,B 0,C 180,E1 -3105.559,E2 -3105.559} C_VEL
LIN {X 0,Y 552.085,Z 87.343,A -85,B 0,C 180,E1 -3108.677,E2 -3108.677} C_VEL
LIN {X 0,Y 552.095,Z 87.34,A -85,B 0,C 180,E1 -3111.408,E2 -3111.408} C_VEL
LIN {X 0,Y 552.101,Z 87.448,A -85,B 0,C 180,E1 -3112.107,E2 -3112.107} C_VEL
LIN {X 0,Y 553.083,Z 93.704,A -85,B 0,C 180,E1 -3113.175,E2 -3113.175} C_VEL
LIN {X 0,Y 552.69,Z 112.462,A -85,B 0,C 180,E1 -3116.197,E2 -3116.197} C_VEL
LIN {X 0,Y 552.648,Z 115.275,A -85,B 0,C 180,E1 -3116.643,E2 -3116.643} C_VEL
LIN {X 0,Y 554.227,Z 123.884,A -85,B 0,C 180,E1 -3116.81,E2 -3116.81} C_VEL
LIN {X 0,Y 553.782,Z 252.214,A -85,B 0,C 180,E1 -3118.519,E2 -3118.519} C_VEL
LIN {X 0,Y 553.574,Z 266.818,A -85,B 0,C 180,E1 -3118.871,E2 -3118.871} C_VEL
LIN {X 0,Y 553.397,Z 280.727,A -85,B 0,C 180,E1 -3119.363,E2 -3119.363} C_VEL
LIN {X 0,Y 553.152,Z 293.673,A -85,B 0,C 180,E1 -3119.971,E2 -3119.971} C_VEL
LIN {X 0,Y 552.899,Z 305.913,A -85,B 0,C 180,E1 -3120.699,E2 -3120.699} C_VEL
LIN {X 0,Y 552.655,Z 317.79,A -85,B 0,C 180,E1 -3121.571,E2 -3121.571} C_VEL
LIN {X 0,Y 552.436,Z 328.589,A -85,B 0,C 180,E1 -3122.537,E2 -3122.537} C_VEL
LIN {X 0,Y 552.201,Z 337.988,A -85,B 0,C 180,E1 -3123.547,E2 -3123.547} C_VEL
LIN {X 0,Y 552.04,Z 346.673,A -85,B 0,C 180,E1 -3124.665,E2 -3124.665} C_VEL
LIN {X 0,Y 551.896,Z 354.889,A -85,B 0,C 180,E1 -3125.951,E2 -3125.951} C_VEL
LIN {X 0,Y 551.817,Z 361.084,A -85,B 0,C 180,E1 -3127.141,E2 -3127.141} C_VEL
LIN {X 0,Y 551.77,Z 366.335,A -85,B 0,C 180,E1 -3128.394,E2 -3128.394} C_VEL
LIN {X 0,Y 551.719,Z 371.071,A -85,B 0,C 180,E1 -3129.882,E2 -3129.882} C_VEL
LIN {X 0,Y 551.712,Z 372.909,A -85,B 0,C 180,E1 -3130.657,E2 -3130.657} C_VEL
LIN {X 0,Y 551.648,Z 375.411,A -85,B 0,C 180,E1 -3132.195,E2 -3132.195} C_VEL
LIN {X 0,Y 551.645,Z 376.436,A -85,B 0,C 180,E1 -3133.722,E2 -3133.722} C_VEL
LIN {X 0,Y 551.669,Z 376.032,A -85,B 0,C 180,E1 -3135.238,E2 -3135.238} C_VEL
LIN {X 0,Y 551.671,Z 374.223,A -85,B 0,C 180,E1 -3136.743,E2 -3136.743} C_VEL
LIN {X 0,Y 551.71,Z 370.987,A -85,B 0,C 180,E1 -3138.239,E2 -3138.239} C_VEL
LIN {X 0,Y 551.763,Z 367.539,A -85,B 0,C 180,E1 -3139.356,E2 -3139.356} C_VEL
LIN {X 0,Y 551.804,Z 361.601,A -85,B 0,C 180,E1 -3140.838,E2 -3140.838} C_VEL
LIN {X 0,Y 551.897,Z 354.932,A -85,B 0,C 180,E1 -3142.131,E2 -3142.131} C_VEL
LIN {X 0,Y 552.064,Z 346.701,A -85,B 0,C 180,E1 -3143.42,E2 -3143.42} C_VEL
LIN {X 0,Y 552.222,Z 338.169,A -85,B 0,C 180,E1 -3144.522,E2 -3144.522} C_VEL
LIN {X 0,Y 552.4,Z 327.886,A -85,B 0,C 180,E1 -3145.621,E2 -3145.621} C_VEL
LIN {X 0,Y 552.65,Z 316.426,A -85,B 0,C 180,E1 -3146.627,E2 -3146.627} C_VEL
LIN {X 0,Y 552.875,Z 305.026,A -85,B 0,C 180,E1 -3147.449,E2 -3147.449} C_VEL
LIN {X 0,Y 553.172,Z 292.522,A -85,B 0,C 180,E1 -3148.179,E2 -3148.179} C_VEL
LIN {X 0,Y 553.436,Z 279.632,A -85,B 0,C 180,E1 -3148.771,E2 -3148.771} C_VEL
LIN {X 0,Y 553.594,Z 265.831,A -85,B 0,C 180,E1 -3149.249,E2 -3149.249} C_VEL
LIN {X 0,Y 553.719,Z 251.309,A -85,B 0,C 180,E1 -3149.59,E2 -3149.59} C_VEL
LIN {X 0,Y 554.154,Z 123.051,A -85,B 0,C 180,E1 -3151.293,E2 -3151.293} C_VEL
LIN {X 0,Y 552.646,Z 115.167,A -85,B 0,C 180,E1 -3151.456,E2 -3151.456} C_VEL
LIN {X 0,Y 553.006,Z 95.868,A -85,B 0,C 180,E1 -3154.555,E2 -3154.555} C_VEL
LIN {X 0,Y 552.897,Z 91.396,A -85,B 0,C 180,E1 -3155.287,E2 -3155.287} C_VEL
LIN {X 0,Y 552.164,Z 87.335,A -85,B 0,C 180,E1 -3156.004,E2 -3156.004} C_VEL
LIN {X 0,Y 552.146,Z 87.329,A -85,B 0,C 180,E1 -3158.785,E2 -3158.785} C_VEL
LIN {X 0,Y 552.128,Z 87.34,A -85,B 0,C 180,E1 -3161.75,E2 -3161.75} C_VEL
LIN {X 0,Y 552.168,Z 87.324,A -85,B 0,C 180,E1 -3164.746,E2 -3164.746} C_VEL
LIN {X 0,Y 552.108,Z 87.338,A -85,B 0,C 180,E1 -3167.787,E2 -3167.787} C_VEL
LIN {X 0,Y 552.102,Z 87.334,A -85,B 0,C 180,E1 -3170.101,E2 -3170.101} C_VEL
LIN {X 0,Y 552.122,Z 87.33,A -85,B 0,C 180,E1 -3172.448,E2 -3172.448} C_VEL
LIN {X 0,Y 552.145,Z 87.337,A -85,B 0,C 180,E1 -3175.358,E2 -3175.358} C_VEL
LIN {X 0,Y 552.105,Z 87.332,A -85,B 0,C 180,E1 -3178.097,E2 -3178.097} C_VEL
LIN {X 0,Y 552.088,Z 87.336,A -85,B 0,C 180,E1 -3180.609,E2 -3180.609} C_VEL
LIN {X 0,Y 552.107,Z 87.34,A -85,B 0,C 180,E1 -3183.185,E2 -3183.185} C_VEL
LIN {X 0,Y 552.1,Z 87.333,A -85,B 0,C 180,E1 -3185.841,E2 -3185.841} C_VEL
LIN {X 0,Y 552.115,Z 87.338,A -85,B 0,C 180,E1 -3189.067,E2 -3189.067} C_VEL
LIN {X 0,Y 552.142,Z 87.329,A -85,B 0,C 180,E1 -3191.442,E2 -3191.442} C_VEL
LIN {X 0,Y 552.097,Z 87.339,A -85,B 0,C 180,E1 -3194.537,E2 -3194.537} C_VEL
LIN {X 0,Y 552.101,Z 87.333,A -85,B 0,C 180,E1 -3197.586,E2 -3197.586} C_VEL
LIN {X 0,Y 552.124,Z 87.338,A -85,B 0,C 180,E1 -3200.477,E2 -3200.477} C_VEL
LIN {X 0,Y 552.111,Z 87.332,A -85,B 0,C 180,E1 -3203.314,E2 -3203.314} C_VEL
LIN {X 0,Y 552.117,Z 87.333,A -85,B 0,C 180,E1 -3205.943,E2 -3205.943} C_VEL
LIN {X 0,Y 552.109,Z 87.338,A -85,B 0,C 180,E1 -3208.544,E2 -3208.544} C_VEL
LIN {X 0,Y 552.111,Z 87.332,A -85,B 0,C 180,E1 -3211.438,E2 -3211.438} C_VEL
LIN {X 0,Y 552.141,Z 87.334,A -85,B 0,C 180,E1 -3214.36,E2 -3214.36} C_VEL
LIN {X 0,Y 552.131,Z 87.33,A -85,B 0,C 180,E1 -3216.763,E2 -3216.763} C_VEL
LIN {X 0,Y 552.117,Z 87.339,A -85,B 0,C 180,E1 -3219.902,E2 -3219.902} C_VEL
LIN {X 0,Y 552.142,Z 87.328,A -85,B 0,C 180,E1 -3222.98,E2 -3222.98} C_VEL
LIN {X 0,Y 552.123,Z 87.336,A -85,B 0,C 180,E1 -3226.007,E2 -3226.007} C_VEL
LIN {X 0,Y 552.164,Z 87.326,A -85,B 0,C 180,E1 -3228.996,E2 -3228.996} C_VEL
LIN {X 0,Y 552.154,Z 87.33,A -85,B 0,C 180,E1 -3231.954,E2 -3231.954} C_VEL
LIN {X 0,Y 552.225,Z 87.319,A -85,B 0,C 180,E1 -3234.892,E2 -3234.892} C_VEL
LIN {X 0,Y 552.213,Z 87.322,A -85,B 0,C 180,E1 -3237.814,E2 -3237.814} C_VEL
LIN {X 0,Y 552.239,Z 87.317,A -85,B 0,C 180,E1 -3240.732,E2 -3240.732} C_VEL
LIN {X 0,Y 552.202,Z 87.324,A -85,B 0,C 180,E1 -3242.92,E2 -3242.92} C_VEL
LIN {X 0,Y 552.192,Z 87.322,A -85,B 0,C 180,E1 -3245.846,E2 -3245.846} C_VEL
LIN {X 0,Y 552.156,Z 87.331,A -85,B 0,C 180,E1 -3248.788,E2 -3248.788} C_VEL
LIN {X 0,Y 552.156,Z 87.326,A -85,B 0,C 180,E1 -3251.753,E2 -3251.753} C_VEL
LIN {X 0,Y 552.131,Z 87.336,A -85,B 0,C 180,E1 -3254.75,E2 -3254.75} C_VEL
LIN {X 0,Y 552.106,Z 87.332,A -85,B 0,C 180,E1 -3257.791,E2 -3257.791} C_VEL
LIN {X 0,Y 552.126,Z 87.331,A -85,B 0,C 180,E1 -3260.103,E2 -3260.103} C_VEL
LIN {X 0,Y 552.091,Z 87.34,A -85,B 0,C 180,E1 -3262.453,E2 -3262.453} C_VEL
LIN {X 0,Y 552.153,Z 87.327,A -85,B 0,C 180,E1 -3265.353,E2 -3265.353} C_VEL
LIN {X 0,Y 552.123,Z 87.334,A -85,B 0,C 180,E1 -3268.099,E2 -3268.099} C_VEL
LIN {X 0,Y 552.099,Z 87.339,A -85,B 0,C 180,E1 -3270.611,E2 -3270.611} C_VEL
LIN {X 0,Y 552.12,Z 87.33,A -85,B 0,C 180,E1 -3273.187,E2 -3273.187} C_VEL
LIN {X 0,Y 552.1,Z 87.336,A -85,B 0,C 180,E1 -3275.844,E2 -3275.844} C_VEL
LIN {X 0,Y 552.119,Z 87.33,A -85,B 0,C 180,E1 -3279.063,E2 -3279.063} C_VEL
LIN {X 0,Y 552.131,Z 87.33,A -85,B 0,C 180,E1 -3281.446,E2 -3281.446} C_VEL
LIN {X 0,Y 552.095,Z 87.335,A -85,B 0,C 180,E1 -3284.534,E2 -3284.534} C_VEL
LIN {X 0,Y 552.13,Z 87.334,A -85,B 0,C 180,E1 -3287.586,E2 -3287.586} C_VEL
LIN {X 0,Y 552.128,Z 87.33,A -85,B 0,C 180,E1 -3290.474,E2 -3290.474} C_VEL
LIN {X 0,Y 552.105,Z 87.336,A -85,B 0,C 180,E1 -3293.319,E2 -3293.319} C_VEL
LIN {X 0,Y 552.125,Z 87.334,A -85,B 0,C 180,E1 -3295.94,E2 -3295.94} C_VEL
LIN {X 0,Y 552.119,Z 87.332,A -85,B 0,C 180,E1 -3298.542,E2 -3298.542} C_VEL
LIN {X 0,Y 552.124,Z 87.339,A -85,B 0,C 180,E1 -3301.44,E2 -3301.44} C_VEL
LIN {X 0,Y 552.129,Z 87.334,A -85,B 0,C 180,E1 -3304.357,E2 -3304.357} C_VEL
LIN {X 0,Y 552.175,Z 87.385,A -85,B 0,C 180,E1 -3304.897,E2 -3304.897} C_VEL
LIN {X 0,Y 553.569,Z 95.353,A -85,B 0,C 180,E1 -3306.079,E2 -3306.079} C_VEL
LIN {X 0,Y 553.149,Z 116.389,A -85,B 0,C 180,E1 -3308.967,E2 -3308.967} C_VEL
LIN {X 0,Y 552.807,Z 137.753,A -85,B 0,C 180,E1 -3311.853,E2 -3311.853} C_VEL
LIN {X 0,Y 552.726,Z 143.183,A -85,B 0,C 180,E1 -3312.581,E2 -3312.581} C_VEL
LIN {X 0,Y 554.203,Z 151.689,A -85,B 0,C 180,E1 -3312.746,E2 -3312.746} C_VEL
LIN {X 0,Y 553.752,Z 281.588,A -85,B 0,C 180,E1 -3314.473,E2 -3314.473} C_VEL
LIN {X 0,Y 553.567,Z 295.794,A -85,B 0,C 180,E1 -3314.811,E2 -3314.811} C_VEL
LIN {X 0,Y 553.376,Z 309.471,A -85,B 0,C 180,E1 -3315.287,E2 -3315.287} C_VEL
LIN {X 0,Y 553.127,Z 323.445,A -85,B 0,C 180,E1 -3315.937,E2 -3315.937} C_VEL
LIN {X 0,Y 552.869,Z 335.948,A -85,B 0,C 180,E1 -3316.68,E2 -3316.68} C_VEL
LIN {X 0,Y 552.654,Z 347.377,A -85,B 0,C 180,E1 -3317.516,E2 -3317.516} C_VEL
LIN {X 0,Y 552.407,Z 358.707,A -85,B 0,C 180,E1 -3318.52,E2 -3318.52} C_VEL
LIN {X 0,Y 552.227,Z 368.329,A -85,B 0,C 180,E1 -3319.552,E2 -3319.552} C_VEL
LIN {X 0,Y 552.071,Z 376.917,A -85,B 0,C 180,E1 -3320.66,E2 -3320.66} C_VEL
LIN {X 0,Y 551.902,Z 385.125,A -85,B 0,C 180,E1 -3321.949,E2 -3321.949} C_VEL
LIN {X 0,Y 551.824,Z 390.868,A -85,B 0,C 180,E1 -3323.052,E2 -3323.052} C_VEL
LIN {X 0,Y 551.792,Z 396.964,A -85,B 0,C 180,E1 -3324.52,E2 -3324.52} C_VEL
LIN {X 0,Y 551.76,Z 400.447,A -85,B 0,C 180,E1 -3325.618,E2 -3325.618} C_VEL
LIN {X 0,Y 551.719,Z 403.834,A -85,B 0,C 180,E1 -3327.08,E2 -3327.08} C_VEL
LIN {X 0,Y 551.641,Z 405.836,A -85,B 0,C 180,E1 -3328.541,E2 -3328.541} C_VEL
LIN {X 0,Y 551.639,Z 406.5,A -85,B 0,C 180,E1 -3330.001,E2 -3330.001} C_VEL
LIN {X 0,Y 551.641,Z 405.835,A -85,B 0,C 180,E1 -3331.461,E2 -3331.461} C_VEL
LIN {X 0,Y 551.72,Z 403.834,A -85,B 0,C 180,E1 -3332.922,E2 -3332.922} C_VEL
LIN {X 0,Y 551.76,Z 400.444,A -85,B 0,C 180,E1 -3334.384,E2 -3334.384} C_VEL
LIN {X 0,Y 551.824,Z 395.563,A -85,B 0,C 180,E1 -3335.849,E2 -3335.849} C_VEL
LIN {X 0,Y 551.836,Z 389.049,A -85,B 0,C 180,E1 -3337.318,E2 -3337.318} C_VEL
LIN {X 0,Y 551.964,Z 381.797,A -85,B 0,C 180,E1 -3338.605,E2 -3338.605} C_VEL
LIN {X 0,Y 552.118,Z 372.813,A -85,B 0,C 180,E1 -3339.896,E2 -3339.896} C_VEL
LIN {X 0,Y 552.332,Z 363.342,A -85,B 0,C 180,E1 -3341.004,E2 -3341.004} C_VEL
LIN {X 0,Y 552.485,Z 352.842,A -85,B 0,C 180,E1 -3342.024,E2 -3342.024} C_VEL
LIN {X 0,Y 552.717,Z 341.261,A -85,B 0,C 180,E1 -3342.951,E2 -3342.951} C_VEL
LIN {X 0,Y 553.015,Z 328.415,A -85,B 0,C 180,E1 -3343.786,E2 -3343.786} C_VEL
LIN {X 0,Y 553.25,Z 315.869,A -85,B 0,C 180,E1 -3344.437,E2 -3344.437} C_VEL
LIN {X 0,Y 553.471,Z 302.714,A -85,B 0,C 180,E1 -3344.966,E2 -3344.966} C_VEL
LIN {X 0,Y 553.647,Z 288.526,A -85,B 0,C 180,E1 -3345.381,E2 -3345.381} C_VEL
LIN {X 0,Y 553.739,Z 274.104,A -85,B 0,C 180,E1 -3345.648,E2 -3345.648} C_VEL
LIN {X 0,Y 554.199,Z 151.974,A -85,B 0,C 180,E1 -3347.25,E2 -3347.25} C_VEL
LIN {X 0,Y 552.737,Z 143.123,A -85,B 0,C 180,E1 -3347.423,E2 -3347.423} C_VEL
LIN {X 0,Y 553.051,Z 120.589,A -85,B 0,C 180,E1 -3350.455,E2 -3350.455} C_VEL
LIN {X 0,Y 553.525,Z 97.984,A -85,B 0,C 180,E1 -3353.546,E2 -3353.546} C_VEL
LIN {X 0,Y 553.408,Z 93.486,A -85,B 0,C 180,E1 -3354.178,E2 -3354.178} C_VEL
LIN {X 0,Y 552.124,Z 87.338,A -85,B 0,C 180,E1 -3355.103,E2 -3355.103} C_VEL
LIN {X 0,Y 552.13,Z 87.332,A -85,B 0,C 180,E1 -3357.275,E2 -3357.275} C_VEL
LIN {X 0,Y 552.121,Z 87.336,A -85,B 0,C 180,E1 -3360.05,E2 -3360.05} C_VEL
LIN {X 0,Y 552.12,Z 87.336,A -85,B 0,C 180,E1 -3362.846,E2 -3362.846} C_VEL
LIN {X 0,Y 552.08,Z 87.337,A -85,B 0,C 180,E1 -3365.439,E2 -3365.439} C_VEL
LIN {X 0,Y 552.105,Z 87.337,A -85,B 0,C 180,E1 -3367.885,E2 -3367.885} C_VEL
LIN {X 0,Y 552.119,Z 87.333,A -85,B 0,C 180,E1 -3370.481,E2 -3370.481} C_VEL
LIN {X 0,Y 552.104,Z 87.336,A -85,B 0,C 180,E1 -3373.481,E2 -3373.481} C_VEL
LIN {X 0,Y 552.119,Z 87.332,A -85,B 0,C 180,E1 -3376.576,E2 -3376.576} C_VEL
LIN {X 0,Y 552.119,Z 87.333,A -85,B 0,C 180,E1 -3379.518,E2 -3379.518} C_VEL
LIN {X 0,Y 552.099,Z 87.333,A -85,B 0,C 180,E1 -3382.335,E2 -3382.335} C_VEL
LIN {X 0,Y 552.092,Z 87.337,A -85,B 0,C 180,E1 -3385.05,E2 -3385.05} C_VEL
LIN {X 0,Y 552.125,Z 87.334,A -85,B 0,C 180,E1 -3387.68,E2 -3387.68} C_VEL
LIN {X 0,Y 552.099,Z 87.334,A -85,B 0,C 180,E1 -3390.233,E2 -3390.233} C_VEL
LIN {X 0,Y 552.108,Z 87.337,A -85,B 0,C 180,E1 -3393.008,E2 -3393.008} C_VEL
LIN {X 0,Y 552.124,Z 87.337,A -85,B 0,C 180,E1 -3395.16,E2 -3395.16} C_VEL
LIN {X 0,Y 552.139,Z 87.33,A -85,B 0,C 180,E1 -3398.336,E2 -3398.336} C_VEL
LIN {X 0,Y 552.162,Z 87.329,A -85,B 0,C 180,E1 -3400.673,E2 -3400.673} C_VEL
LIN {X 0,Y 552.115,Z 87.33,A -85,B 0,C 180,E1 -3403.735,E2 -3403.735} C_VEL
LIN {X 0,Y 552.14,Z 87.329,A -85,B 0,C 180,E1 -3406.003,E2 -3406.003} C_VEL
LIN {X 0,Y 552.171,Z 87.327,A -85,B 0,C 180,E1 -3408.992,E2 -3408.992} C_VEL
LIN {X 0,Y 552.155,Z 87.328,A -85,B 0,C 180,E1 -3411.949,E2 -3411.949} C_VEL
LIN {X 0,Y 552.226,Z 87.32,A -85,B 0,C 180,E1 -3414.887,E2 -3414.887} C_VEL
LIN {X 0,Y 552.228,Z 87.319,A -85,B 0,C 180,E1 -3417.81,E2 -3417.81} C_VEL
LIN {X 0,Y 552.24,Z 87.315,A -85,B 0,C 180,E1 -3420.727,E2 -3420.727} C_VEL
LIN {X 0,Y 552.201,Z 87.321,A -85,B 0,C 180,E1 -3422.916,E2 -3422.916} C_VEL
LIN {X 0,Y 552.195,Z 87.328,A -85,B 0,C 180,E1 -3425.841,E2 -3425.841} C_VEL
LIN {X 0,Y 552.142,Z 87.327,A -85,B 0,C 180,E1 -3428.783,E2 -3428.783} C_VEL
LIN {X 0,Y 552.163,Z 87.333,A -85,B 0,C 180,E1 -3431.748,E2 -3431.748} C_VEL
LIN {X 0,Y 552.128,Z 87.33,A -85,B 0,C 180,E1 -3434.746,E2 -3434.746} C_VEL
LIN {X 0,Y 552.093,Z 87.339,A -85,B 0,C 180,E1 -3437.786,E2 -3437.786} C_VEL
LIN {X 0,Y 552.121,Z 87.33,A -85,B 0,C 180,E1 -3440.098,E2 -3440.098} C_VEL
LIN {X 0,Y 552.085,Z 87.336,A -85,B 0,C 180,E1 -3442.448,E2 -3442.448} C_VEL
LIN {X 0,Y 552.099,Z 87.339,A -85,B 0,C 180,E1 -3445.336,E2 -3445.336} C_VEL
LIN {X 0,Y 552.083,Z 87.335,A -85,B 0,C 180,E1 -3448.096,E2 -3448.096} C_VEL
LIN {X 0,Y 552.087,Z 87.335,A -85,B 0,C 180,E1 -3450.606,E2 -3450.606} C_VEL
LIN {X 0,Y 552.093,Z 87.337,A -85,B 0,C 180,E1 -3453.183,E2 -3453.183} C_VEL
LIN {X 0,Y 552.076,Z 87.334,A -85,B 0,C 180,E1 -3453.762,E2 -3453.762} C_VEL
LIN {X 0,Y 551.435,Z 87.418,A -85,B 0,C 180,E1 -3454.371,E2 -3454.371} C_VEL
LIN {X 0,Y 548.624,Z 87.773,A -85,B 0,C 180,E1 -3455.359,E2 -3455.359} C_VEL
LIN {X 0,Y 546.216,Z 88.076,A -85,B 0,C 180,E1 -3456.155,E2 -3456.155} C_VEL
LIN {X 0,Y 545.151,Z 88.206,A -85,B 0,C 180,E1 -3456.769,E2 -3456.769} C_VEL
LIN {X 0,Y 545.048,Z 88.215,A -85,B 0,C 180,E1 -3456.977,E2 -3456.977} C_VEL
LIN {X 0,Y 545.046,Z 88.216,A -85,B 0,C 180,E1 -3460.139,E2 -3460.139} C_VEL
LIN {X 0,Y 545.06,Z 88.213,A -85,B 0,C 180,E1 -3463.103,E2 -3463.103} C_VEL
LIN {X 0,Y 545.028,Z 88.222,A -85,B 0,C 180,E1 -3466.223,E2 -3466.223} C_VEL
LIN {X 0,Y 545.049,Z 88.219,A -85,B 0,C 180,E1 -3468.881,E2 -3468.881} C_VEL
LIN {X 0,Y 545.048,Z 88.221,A -85,B 0,C 180,E1 -3471.761,E2 -3471.761} C_VEL
LIN {X 0,Y 545.067,Z 88.269,A -85,B 0,C 180,E1 -3471.921,E2 -3471.921} C_VEL
LIN {X 0,Y 546.07,Z 94.068,A -85,B 0,C 180,E1 -3472.928,E2 -3472.928} C_VEL
LIN {X 0,Y 545.841,Z 109.75,A -85,B 0,C 180,E1 -3475.491,E2 -3475.491} C_VEL
LIN {X 0,Y 545.695,Z 115.437,A -85,B 0,C 180,E1 -3476.409,E2 -3476.409} C_VEL
LIN {X 0,Y 547.457,Z 125.119,A -85,B 0,C 180,E1 -3476.604,E2 -3476.604} C_VEL
LIN {X 0,Y 546.947,Z 252.131,A -85,B 0,C 180,E1 -3478.316,E2 -3478.316} C_VEL
LIN {X 0,Y 546.737,Z 266.231,A -85,B 0,C 180,E1 -3478.653,E2 -3478.653} C_VEL
LIN {X 0,Y 546.558,Z 279.529,A -85,B 0,C 180,E1 -3479.118,E2 -3479.118} C_VEL
LIN {X 0,Y 546.287,Z 292.318,A -85,B 0,C 180,E1 -3479.708,E2 -3479.708} C_VEL
LIN {X 0,Y 546.015,Z 304.167,A -85,B 0,C 180,E1 -3480.399,E2 -3480.399} C_VEL
LIN {X 0,Y 545.725,Z 316.283,A -85,B 0,C 180,E1 -3481.273,E2 -3481.273} C_VEL
LIN {X 0,Y 545.487,Z 327.467,A -85,B 0,C 180,E1 -3482.261,E2 -3482.261} C_VEL
LIN {X 0,Y 545.212,Z 337.978,A -85,B 0,C 180,E1 -3483.387,E2 -3483.387} C_VEL
LIN {X 0,Y 545.001,Z 346.572,A -85,B 0,C 180,E1 -3484.502,E2 -3484.502} C_VEL
LIN {X 0,Y 544.851,Z 354.911,A -85,B 0,C 180,E1 -3485.816,E2 -3485.816} C_VEL
LIN {X 0,Y 544.729,Z 362.027,A -85,B 0,C 180,E1 -3487.228,E2 -3487.228} C_VEL
LIN {X 0,Y 544.679,Z 366.263,A -85,B 0,C 180,E1 -3488.27,E2 -3488.27} C_VEL
LIN {X 0,Y 544.645,Z 370.551,A -85,B 0,C 180,E1 -3489.609,E2 -3489.609} C_VEL
LIN {X 0,Y 544.615,Z 372.516,A -85,B 0,C 180,E1 -3490.395,E2 -3490.395} C_VEL
LIN {X 0,Y 544.542,Z 375.236,A -85,B 0,C 180,E1 -3491.955,E2 -3491.955} C_VEL
LIN {X 0,Y 544.561,Z 376.439,A -85,B 0,C 180,E1 -3493.504,E2 -3493.504} C_VEL
LIN {X 0,Y 544.561,Z 376.22,A -85,B 0,C 180,E1 -3495.041,E2 -3495.041} C_VEL
LIN {X 0,Y 544.597,Z 374.603,A -85,B 0,C 180,E1 -3496.567,E2 -3496.567} C_VEL
LIN {X 0,Y 544.609,Z 371.582,A -85,B 0,C 180,E1 -3498.083,E2 -3498.083} C_VEL
LIN {X 0,Y 544.661,Z 367.096,A -85,B 0,C 180,E1 -3499.591,E2 -3499.591} C_VEL
LIN {X 0,Y 544.718,Z 362.647,A -85,B 0,C 180,E1 -3500.718,E2 -3500.718} C_VEL
LIN {X 0,Y 544.83,Z 356.236,A -85,B 0,C 180,E1 -3502.028,E2 -3502.028} C_VEL
LIN {X 0,Y 544.986,Z 348.308,A -85,B 0,C 180,E1 -3503.334,E2 -3503.334} C_VEL
LIN {X 0,Y 545.147,Z 340.052,A -85,B 0,C 180,E1 -3504.45,E2 -3504.45} C_VEL
LIN {X 0,Y 545.355,Z 330.156,A -85,B 0,C 180,E1 -3505.564,E2 -3505.564} C_VEL
LIN {X 0,Y 545.641,Z 319.165,A -85,B 0,C 180,E1 -3506.584,E2 -3506.584} C_VEL
LIN {X 0,Y 545.928,Z 306.907,A -85,B 0,C 180,E1 -3507.509,E2 -3507.509} C_VEL
LIN {X 0,Y 546.258,Z 294.79,A -85,B 0,C 180,E1 -3508.248,E2 -3508.248} C_VEL
LIN {X 0,Y 546.503,Z 281.413,A -85,B 0,C 180,E1 -3508.894,E2 -3508.894} C_VEL
LIN {X 0,Y 546.706,Z 267.403,A -85,B 0,C 180,E1 -3509.401,E2 -3509.401} C_VEL
LIN {X 0,Y 546.856,Z 253.595,A -85,B 0,C 180,E1 -3509.746,E2 -3509.746} C_VEL
LIN {X 0,Y 547.001,Z 226.395,A -85,B 0,C 180,E1 -3510.137,E2 -3510.137} C_VEL
LIN {X 0,Y 547.369,Z 123.914,A -85,B 0,C 180,E1 -3511.505,E2 -3511.505} C_VEL
LIN {X 0,Y 545.718,Z 115.373,A -85,B 0,C 180,E1 -3511.682,E2 -3511.682} C_VEL
LIN {X 0,Y 546.098,Z 96.198,A -85,B 0,C 180,E1 -3514.797,E2 -3514.797} C_VEL
LIN {X 0,Y 545.988,Z 92.851,A -85,B 0,C 180,E1 -3515.354,E2 -3515.354} C_VEL
LIN {X 0,Y 545.116,Z 88.212,A -85,B 0,C 180,E1 -3516.198,E2 -3516.198} C_VEL
LIN {X 0,Y 545.102,Z 88.207,A -85,B 0,C 180,E1 -3518.899,E2 -3518.899} C_VEL
LIN {X 0,Y 545.1,Z 88.215,A -85,B 0,C 180,E1 -3521.904,E2 -3521.904} C_VEL
LIN {X 0,Y 545.104,Z 88.205,A -85,B 0,C 180,E1 -3524.942,E2 -3524.942} C_VEL
LIN {X 0,Y 545.067,Z 88.212,A -85,B 0,C 180,E1 -3528.025,E2 -3528.025} C_VEL
LIN {X 0,Y 545.067,Z 88.209,A -85,B 0,C 180,E1 -3530.372,E2 -3530.372} C_VEL
LIN {X 0,Y 545.112,Z 88.21,A -85,B 0,C 180,E1 -3533.557,E2 -3533.557} C_VEL
LIN {X 0,Y 545.077,Z 88.209,A -85,B 0,C 180,E1 -3535.999,E2 -3535.999} C_VEL
LIN {X 0,Y 545.072,Z 88.211,A -85,B 0,C 180,E1 -3538.753,E2 -3538.753} C_VEL
LIN {X 0,Y 545.051,Z 88.213,A -85,B 0,C 180,E1 -3541.685,E2 -3541.685} C_VEL
LIN {X 0,Y 545.063,Z 88.212,A -85,B 0,C 180,E1 -3544.563,E2 -3544.563} C_VEL
LIN {X 0,Y 545.058,Z 88.215,A -85,B 0,C 180,E1 -3547.301,E2 -3547.301} C_VEL
LIN {X 0,Y 545.117,Z 88.203,A -85,B 0,C 180,E1 -3550.136,E2 -3550.136} C_VEL
LIN {X 0,Y 545.061,Z 88.214,A -85,B 0,C 180,E1 -3553.107,E2 -3553.107} C_VEL
LIN {X 0,Y 545.053,Z 88.211,A -85,B 0,C 180,E1 -3555.876,E2 -3555.876} C_VEL
LIN {X 0,Y 545.094,Z 88.211,A -85,B 0,C 180,E1 -3558.891,E2 -3558.891} C_VEL
LIN {X 0,Y 545.028,Z 88.214,A -85,B 0,C 180,E1 -3561.765,E2 -3561.765} C_VEL
LIN {X 0,Y 545.047,Z 88.22,A -85,B 0,C 180,E1 -3564.537,E2 -3564.537} C_VEL
LIN {X 0,Y 545.059,Z 88.21,A -85,B 0,C 180,E1 -3567.215,E2 -3567.215} C_VEL
LIN {X 0,Y 545.076,Z 88.21,A -85,B 0,C 180,E1 -3569.815,E2 -3569.815} C_VEL
LIN {X 0,Y 545.08,Z 88.209,A -85,B 0,C 180,E1 -3572.827,E2 -3572.827} C_VEL
LIN {X 0,Y 545.049,Z 88.214,A -85,B 0,C 180,E1 -3575.634,E2 -3575.634} C_VEL
LIN {X 0,Y 545.078,Z 88.215,A -85,B 0,C 180,E1 -3578.173,E2 -3578.173} C_VEL
LIN {X 0,Y 545.068,Z 88.209,A -85,B 0,C 180,E1 -3581.198,E2 -3581.198} C_VEL
LIN {X 0,Y 545.063,Z 88.214,A -85,B 0,C 180,E1 -3583.524,E2 -3583.524} C_VEL
LIN {X 0,Y 545.08,Z 88.216,A -85,B 0,C 180,E1 -3585.823,E2 -3585.823} C_VEL
LIN {X 0,Y 545.118,Z 88.203,A -85,B 0,C 180,E1 -3588.852,E2 -3588.852} C_VEL
LIN {X 0,Y 545.124,Z 88.207,A -85,B 0,C 180,E1 -3591.85,E2 -3591.85} C_VEL
LIN {X 0,Y 545.2,Z 88.193,A -85,B 0,C 180,E1 -3594.826,E2 -3594.826} C_VEL
LIN {X 0,Y 545.185,Z 88.198,A -85,B 0,C 180,E1 -3597.786,E2 -3597.786} C_VEL
LIN {X 0,Y 545.208,Z 88.193,A -85,B 0,C 180,E1 -3600.741,E2 -3600.741} C_VEL
LIN {X 0,Y 545.168,Z 88.201,A -85,B 0,C 180,E1 -3602.958,E2 -3602.958} C_VEL
LIN {X 0,Y 545.163,Z 88.197,A -85,B 0,C 180,E1 -3605.922,E2 -3605.922} C_VEL
LIN {X 0,Y 545.114,Z 88.21,A -85,B 0,C 180,E1 -3608.902,E2 -3608.902} C_VEL
LIN {X 0,Y 545.128,Z 88.201,A -85,B 0,C 180,E1 -3611.906,E2 -3611.906} C_VEL
LIN {X 0,Y 545.08,Z 88.216,A -85,B 0,C 180,E1 -3614.946,E2 -3614.946} C_VEL
LIN {X 0,Y 545.074,Z 88.209,A -85,B 0,C 180,E1 -3618.028,E2 -3618.028} C_VEL
LIN {X 0,Y 545.091,Z 88.21,A -85,B 0,C 180,E1 -3620.374,E2 -3620.374} C_VEL
LIN {X 0,Y 545.087,Z 88.206,A -85,B 0,C 180,E1 -3623.561,E2 -3623.561} C_VEL
LIN {X 0,Y 545.085,Z 88.209,A -85,B 0,C 180,E1 -3626.002,E2 -3626.002} C_VEL
LIN {X 0,Y 545.087,Z 88.211,A -85,B 0,C 180,E1 -3628.75,E2 -3628.75} C_VEL
LIN {X 0,Y 545.056,Z 88.211,A -85,B 0,C 180,E1 -3631.681,E2 -3631.681} C_VEL
LIN {X 0,Y 545.074,Z 88.213,A -85,B 0,C 180,E1 -3634.565,E2 -3634.565} C_VEL
LIN {X 0,Y 545.036,Z 88.213,A -85,B 0,C 180,E1 -3637.306,E2 -3637.306} C_VEL
LIN {X 0,Y 545.064,Z 88.218,A -85,B 0,C 180,E1 -3640.144,E2 -3640.144} C_VEL
LIN {X 0,Y 545.077,Z 88.208,A -85,B 0,C 180,E1 -3643.108,E2 -3643.108} C_VEL
LIN {X 0,Y 545.049,Z 88.216,A -85,B 0,C 180,E1 -3646.228,E2 -3646.228} C_VEL
LIN {X 0,Y 545.085,Z 88.207,A -85,B 0,C 180,E1 -3648.887,E2 -3648.887} C_VEL
LIN {X 0,Y 545.052,Z 88.22,A -85,B 0,C 180,E1 -3651.764,E2 -3651.764} C_VEL
LIN {X 0,Y 545.035,Z 88.213,A -85,B 0,C 180,E1 -3654.533,E2 -3654.533} C_VEL
LIN {X 0,Y 545.066,Z 88.213,A -85,B 0,C 180,E1 -3657.213,E2 -3657.213} C_VEL
LIN {X 0,Y 545.061,Z 88.216,A -85,B 0,C 180,E1 -3659.812,E2 -3659.812} C_VEL
LIN {X 0,Y 545.081,Z 88.21,A -85,B 0,C 180,E1 -3662.345,E2 -3662.345} C_VEL
LIN {X 0,Y 545.109,Z 88.274,A -85,B 0,C 180,E1 -3664.699,E2 -3664.699} C_VEL
LIN {X 0,Y 546.621,Z 96.245,A -85,B 0,C 180,E1 -3665.905,E2 -3665.905} C_VEL
LIN {X 0,Y 546.286,Z 114.774,A -85,B 0,C 180,E1 -3668.492,E2 -3668.492} C_VEL
LIN {X 0,Y 545.881,Z 136.136,A -85,B 0,C 180,E1 -3671.42,E2 -3671.42} C_VEL
LIN {X 0,Y 545.749,Z 143.079,A -85,B 0,C 180,E1 -3672.356,E2 -3672.356} C_VEL
LIN {X 0,Y 547.419,Z 152.762,A -85,B 0,C 180,E1 -3672.542,E2 -3672.542} C_VEL
LIN {X 0,Y 546.916,Z 281.343,A -85,B 0,C 180,E1 -3674.274,E2 -3674.274} C_VEL
LIN {X 0,Y 546.727,Z 295.123,A -85,B 0,C 180,E1 -3674.603,E2 -3674.603} C_VEL
LIN {X 0,Y 546.495,Z 309.251,A -85,B 0,C 180,E1 -3675.097,E2 -3675.097} C_VEL
LIN {X 0,Y 546.193,Z 323.23,A -85,B 0,C 180,E1 -3675.755,E2 -3675.755} C_VEL
LIN {X 0,Y 545.898,Z 335.737,A -85,B 0,C 180,E1 -3676.507,E2 -3676.507} C_VEL
LIN {X 0,Y 545.642,Z 347.168,A -85,B 0,C 180,E1 -3677.353,E2 -3677.353} C_VEL
LIN {X 0,Y 545.459,Z 357.787,A -85,B 0,C 180,E1 -3678.303,E2 -3678.303} C_VEL
LIN {X 0,Y 545.169,Z 368.126,A -85,B 0,C 180,E1 -3679.416,E2 -3679.416} C_VEL
LIN {X 0,Y 545.004,Z 376.75,A -85,B 0,C 180,E1 -3680.538,E2 -3680.538} C_VEL
LIN {X 0,Y 544.847,Z 385.009,A -85,B 0,C 180,E1 -3681.844,E2 -3681.844} C_VEL
LIN {X 0,Y 544.737,Z 390.789,A -85,B 0,C 180,E1 -3682.961,E2 -3682.961} C_VEL
LIN {X 0,Y 544.732,Z 395.527,A -85,B 0,C 180,E1 -3684.077,E2 -3684.077} C_VEL
LIN {X 0,Y 544.654,Z 400.434,A -85,B 0,C 180,E1 -3685.561,E2 -3685.561} C_VEL
LIN {X 0,Y 544.646,Z 403.833,A -85,B 0,C 180,E1 -3687.042,E2 -3687.042} C_VEL
LIN {X 0,Y 544.542,Z 405.836,A -85,B 0,C 180,E1 -3688.522,E2 -3688.522} C_VEL
LIN {X 0,Y 544.539,Z 406.5,A -85,B 0,C 180,E1 -3690.001,E2 -3690.001} C_VEL
LIN {X 0,Y 544.542,Z 405.836,A -85,B 0,C 180,E1 -3691.48,E2 -3691.48} C_VEL
LIN {X 0,Y 544.647,Z 403.833,A -85,B 0,C 180,E1 -3692.96,E2 -3692.96} C_VEL
LIN {X 0,Y 544.655,Z 400.431,A -85,B 0,C 180,E1 -3694.441,E2 -3694.441} C_VEL
LIN {X 0,Y 544.737,Z 395.516,A -85,B 0,C 180,E1 -3695.925,E2 -3695.925} C_VEL
LIN {X 0,Y 544.74,Z 390.775,A -85,B 0,C 180,E1 -3697.041,E2 -3697.041} C_VEL
LIN {X 0,Y 544.875,Z 383.901,A -85,B 0,C 180,E1 -3698.344,E2 -3698.344} C_VEL
LIN {X 0,Y 545.014,Z 375.367,A -85,B 0,C 180,E1 -3699.651,E2 -3699.651} C_VEL
LIN {X 0,Y 545.228,Z 366.464,A -85,B 0,C 180,E1 -3700.773,E2 -3700.773} C_VEL
LIN {X 0,Y 545.452,Z 355.679,A -85,B 0,C 180,E1 -3701.898,E2 -3701.898} C_VEL
LIN {X 0,Y 545.705,Z 344.768,A -85,B 0,C 180,E1 -3702.837,E2 -3702.837} C_VEL
LIN {X 0,Y 545.962,Z 332.826,A -85,B 0,C 180,E1 -3703.683,E2 -3703.683} C_VEL
LIN {X 0,Y 546.288,Z 319.609,A -85,B 0,C 180,E1 -3704.435,E2 -3704.435} C_VEL
LIN {X 0,Y 546.589,Z 307.204,A -85,B 0,C 180,E1 -3704.985,E2 -3704.985} C_VEL
LIN {X 0,Y 546.718,Z 293.176,A -85,B 0,C 180,E1 -3705.453,E2 -3705.453} C_VEL
LIN {X 0,Y 546.908,Z 279.883,A -85,B 0,C 180,E1 -3705.752,E2 -3705.752} C_VEL
LIN {X 0,Y 547.422,Z 152.609,A -85,B 0,C 180,E1 -3707.459,E2 -3707.459} C_VEL
LIN {X 0,Y 545.757,Z 142.903,A -85,B 0,C 180,E1 -3707.654,E2 -3707.654} C_VEL
LIN {X 0,Y 546.145,Z 120.378,A -85,B 0,C 180,E1 -3710.726,E2 -3710.726} C_VEL
LIN {X 0,Y 546.632,Z 99.346,A -85,B 0,C 180,E1 -3713.643,E2 -3713.643} C_VEL
LIN {X 0,Y 546.465,Z 94.73,A -85,B 0,C 180,E1 -3714.303,E2 -3714.303} C_VEL
LIN {X 0,Y 545.067,Z 88.216,A -85,B 0,C 180,E1 -3715.301,E2 -3715.301} C_VEL
LIN {X 0,Y 545.083,Z 88.209,A -85,B 0,C 180,E1 -3717.657,E2 -3717.657} C_VEL
LIN {X 0,Y 545.066,Z 88.218,A -85,B 0,C 180,E1 -3720.243,E2 -3720.243} C_VEL
LIN {X 0,Y 545.084,Z 88.211,A -85,B 0,C 180,E1 -3723.061,E2 -3723.061} C_VEL
LIN {X 0,Y 545.035,Z 88.216,A -85,B 0,C 180,E1 -3725.672,E2 -3725.672} C_VEL
LIN {X 0,Y 545.062,Z 88.219,A -85,B 0,C 180,E1 -3728.238,E2 -3728.238} C_VEL
LIN {X 0,Y 545.092,Z 88.205,A -85,B 0,C 180,E1 -3731.115,E2 -3731.115} C_VEL
LIN {X 0,Y 545.05,Z 88.218,A -85,B 0,C 180,E1 -3734.131,E2 -3734.131} C_VEL
LIN {X 0,Y 545.091,Z 88.207,A -85,B 0,C 180,E1 -3736.893,E2 -3736.893} C_VEL
LIN {X 0,Y 545.076,Z 88.215,A -85,B 0,C 180,E1 -3739.857,E2 -3739.857} C_VEL
LIN {X 0,Y 545.077,Z 88.21,A -85,B 0,C 180,E1 -3743.074,E2 -3743.074} C_VEL
LIN {X 0,Y 545.061,Z 88.21,A -85,B 0,C 180,E1 -3746.326,E2 -3746.326} C_VEL
LIN {X 0,Y 545.075,Z 88.211,A -85,B 0,C 180,E1 -3748.951,E2 -3748.951} C_VEL
LIN {X 0,Y 545.086,Z 88.211,A -85,B 0,C 180,E1 -3751.505,E2 -3751.505} C_VEL
LIN {X 0,Y 545.117,Z 88.208,A -85,B 0,C 180,E1 -3754.819,E2 -3754.819} C_VEL
LIN {X 0,Y 545.045,Z 88.218,A -85,B 0,C 180,E1 -3757.241,E2 -3757.241} C_VEL
LIN {X 0,Y 545.128,Z 88.202,A -85,B 0,C 180,E1 -3760.413,E2 -3760.413} C_VEL
LIN {X 0,Y 545.066,Z 88.208,A -85,B 0,C 180,E1 -3763.519,E2 -3763.519} C_VEL
LIN {X 0,Y 545.094,Z 88.206,A -85,B 0,C 180,E1 -3765.818,E2 -3765.818} C_VEL
LIN {X 0,Y 545.127,Z 88.207,A -85,B 0,C 180,E1 -3768.847,E2 -3768.847} C_VEL
LIN {X 0,Y 545.103,Z 88.206,A -85,B 0,C 180,E1 -3771.845,E2 -3771.845} C_VEL
LIN {X 0,Y 545.201,Z 88.195,A -85,B 0,C 180,E1 -3774.821,E2 -3774.821} C_VEL
LIN {X 0,Y 545.2,Z 88.194,A -85,B 0,C 180,E1 -3777.781,E2 -3777.781} C_VEL
LIN {X 0,Y 545.212,Z 88.19,A -85,B 0,C 180,E1 -3780.736,E2 -3780.736} C_VEL
LIN {X 0,Y 545.169,Z 88.197,A -85,B 0,C 180,E1 -3782.953,E2 -3782.953} C_VEL
LIN {X 0,Y 545.165,Z 88.204,A -85,B 0,C 180,E1 -3785.917,E2 -3785.917} C_VEL
LIN {X 0,Y 545.103,Z 88.204,A -85,B 0,C 180,E1 -3788.898,E2 -3788.898} C_VEL
LIN {X 0,Y 545.106,Z 88.21,A -85,B 0,C 180,E1 -3791.902,E2 -3791.902} C_VEL
LIN {X 0,Y 545.081,Z 88.209,A -85,B 0,C 180,E1 -3794.941,E2 -3794.941} C_VEL
LIN {X 0,Y 545.058,Z 88.212,A -85,B 0,C 180,E1 -3798.023,E2 -3798.023} C_VEL
LIN {X 0,Y 545.087,Z 88.206,A -85,B 0,C 180,E1 -3800.369,E2 -3800.369} C_VEL
LIN {X 0,Y 545.069,Z 88.214,A -85,B 0,C 180,E1 -3803.556,E2 -3803.556} C_VEL
LIN {X 0,Y 545.061,Z 88.209,A -85,B 0,C 180,E1 -3805.998,E2 -3805.998} C_VEL
LIN {X 0,Y 545.065,Z 88.214,A -85,B 0,C 180,E1 -3808.742,E2 -3808.742} C_VEL
LIN {X 0,Y 545.046,Z 88.213,A -85,B 0,C 180,E1 -3811.675,E2 -3811.675} C_VEL
LIN {X 0,Y 545.046,Z 88.215,A -85,B 0,C 180,E1 -3814.561,E2 -3814.561} C_VEL
LIN {X 0,Y 545.048,Z 88.215,A -85,B 0,C 180,E1 -3816.977,E2 -3816.977} C_VEL
LIN {X 0,Y 544.335,Z 88.301,A -85,B 0,C 180,E1 -3817.593,E2 -3817.593} C_VEL
LIN {X 0,Y 541.462,Z 88.664,A -85,B 0,C 180,E1 -3818.594,E2 -3818.594} C_VEL
LIN {X 0,Y 539.072,Z 88.959,A -85,B 0,C 180,E1 -3819.4,E2 -3819.4} C_VEL
LIN {X 0,Y 538.065,Z 89.085,A -85,B 0,C 180,E1 -3820.022,E2 -3820.022} C_VEL
LIN {X 0,Y 537.992,Z 89.092,A -85,B 0,C 180,E1 -3820.233,E2 -3820.233} C_VEL
LIN {X 0,Y 538.008,Z 89.093,A -85,B 0,C 180,E1 -3822.984,E2 -3822.984} C_VEL
LIN {X 0,Y 537.982,Z 89.099,A -85,B 0,C 180,E1 -3826.181,E2 -3826.181} C_VEL
LIN {X 0,Y 537.999,Z 89.096,A -85,B 0,C 180,E1 -3829.253,E2 -3829.253} C_VEL
LIN {X 0,Y 538.005,Z 89.105,A -85,B 0,C 180,E1 -3831.727,E2 -3831.727} C_VEL
LIN {X 0,Y 539.161,Z 95.899,A -85,B 0,C 180,E1 -3832.921,E2 -3832.921} C_VEL
LIN {X 0,Y 538.863,Z 111.37,A -85,B 0,C 180,E1 -3835.475,E2 -3835.475} C_VEL
LIN {X 0,Y 538.76,Z 115.62,A -85,B 0,C 180,E1 -3836.171,E2 -3836.171} C_VEL
LIN {X 0,Y 540.69,Z 125.542,A -85,B 0,C 180,E1 -3836.382,E2 -3836.382} C_VEL
LIN {X 0,Y 540.114,Z 252.415,A -85,B 0,C 180,E1 -3838.114,E2 -3838.114} C_VEL
LIN {X 0,Y 539.91,Z 266.503,A -85,B 0,C 180,E1 -3838.457,E2 -3838.457} C_VEL
LIN {X 0,Y 539.698,Z 280.349,A -85,B 0,C 180,E1 -3838.951,E2 -3838.951} C_VEL
LIN {X 0,Y 539.398,Z 293.334,A -85,B 0,C 180,E1 -3839.567,E2 -3839.567} C_VEL
LIN {X 0,Y 539.081,Z 305.565,A -85,B 0,C 180,E1 -3840.302,E2 -3840.302} C_VEL
LIN {X 0,Y 538.787,Z 316.899,A -85,B 0,C 180,E1 -3841.142,E2 -3841.142} C_VEL
LIN {X 0,Y 538.494,Z 328.08,A -85,B 0,C 180,E1 -3842.147,E2 -3842.147} C_VEL
LIN {X 0,Y 538.201,Z 337.961,A -85,B 0,C 180,E1 -3843.222,E2 -3843.222} C_VEL
LIN {X 0,Y 537.971,Z 347.364,A -85,B 0,C 180,E1 -3844.461,E2 -3844.461} C_VEL
LIN {X 0,Y 537.794,Z 355.006,A -85,B 0,C 180,E1 -3845.691,E2 -3845.691} C_VEL
LIN {X 0,Y 537.676,Z 361.21,A -85,B 0,C 180,E1 -3846.912,E2 -3846.912} C_VEL
LIN {X 0,Y 537.621,Z 366.235,A -85,B 0,C 180,E1 -3848.135,E2 -3848.135} C_VEL
LIN {X 0,Y 537.572,Z 370.122,A -85,B 0,C 180,E1 -3849.329,E2 -3849.329} C_VEL
LIN {X 0,Y 537.561,Z 372.508,A -85,B 0,C 180,E1 -3850.261,E2 -3850.261} C_VEL
LIN {X 0,Y 537.442,Z 375.13,A -85,B 0,C 180,E1 -3851.708,E2 -3851.708} C_VEL
LIN {X 0,Y 537.496,Z 376.162,A -85,B 0,C 180,E1 -3852.636,E2 -3852.636} C_VEL
LIN {X 0,Y 537.444,Z 376.744,A -85,B 0,C 180,E1 -3854.06,E2 -3854.06} C_VEL
LIN {X 0,Y 537.512,Z 376.006,A -85,B 0,C 180,E1 -3855.615,E2 -3855.615} C_VEL
LIN {X 0,Y 537.518,Z 373.873,A -85,B 0,C 180,E1 -3857.156,E2 -3857.156} C_VEL
LIN {X 0,Y 537.567,Z 370.315,A -85,B 0,C 180,E1 -3858.69,E2 -3858.69} C_VEL
LIN {X 0,Y 537.609,Z 365.256,A -85,B 0,C 180,E1 -3860.214,E2 -3860.214} C_VEL
LIN {X 0,Y 537.683,Z 360.364,A -85,B 0,C 180,E1 -3861.354,E2 -3861.354} C_VEL
LIN {X 0,Y 537.849,Z 353.344,A -85,B 0,C 180,E1 -3862.68,E2 -3862.68} C_VEL
LIN {X 0,Y 538.018,Z 344.707,A -85,B 0,C 180,E1 -3864,E2 -3864} C_VEL
LIN {X 0,Y 538.277,Z 335.691,A -85,B 0,C 180,E1 -3865.131,E2 -3865.131} C_VEL
LIN {X 0,Y 538.567,Z 324.83,A -85,B 0,C 180,E1 -3866.258,E2 -3866.258} C_VEL
LIN {X 0,Y 538.852,Z 313.817,A -85,B 0,C 180,E1 -3867.196,E2 -3867.196} C_VEL
LIN {X 0,Y 539.149,Z 301.711,A -85,B 0,C 180,E1 -3868.038,E2 -3868.038} C_VEL
LIN {X 0,Y 539.517,Z 288.165,A -85,B 0,C 180,E1 -3868.786,E2 -3868.786} C_VEL
LIN {X 0,Y 539.778,Z 275.032,A -85,B 0,C 180,E1 -3869.346,E2 -3869.346} C_VEL
LIN {X 0,Y 539.98,Z 260.771,A -85,B 0,C 180,E1 -3869.789,E2 -3869.789} C_VEL
LIN {X 0,Y 540.077,Z 246.856,A -85,B 0,C 180,E1 -3870.069,E2 -3870.069} C_VEL
LIN {X 0,Y 540.683,Z 125.38,A -85,B 0,C 180,E1 -3871.71,E2 -3871.71} C_VEL
LIN {X 0,Y 538.773,Z 115.469,A -85,B 0,C 180,E1 -3871.933,E2 -3871.933} C_VEL
LIN {X 0,Y 539.164,Z 97.662,A -85,B 0,C 180,E1 -3874.859,E2 -3874.859} C_VEL
LIN {X 0,Y 539.057,Z 94.312,A -85,B 0,C 180,E1 -3875.423,E2 -3875.423} C_VEL
LIN {X 0,Y 538.082,Z 89.087,A -85,B 0,C 180,E1 -3876.373,E2 -3876.373} C_VEL
LIN {X 0,Y 538.051,Z 89.086,A -85,B 0,C 180,E1 -3879.017,E2 -3879.017} C_VEL
LIN {X 0,Y 538.052,Z 89.091,A -85,B 0,C 180,E1 -3882.062,E2 -3882.062} C_VEL
LIN {X 0,Y 538.044,Z 89.086,A -85,B 0,C 180,E1 -3885.143,E2 -3885.143} C_VEL
LIN {X 0,Y 538.053,Z 89.091,A -85,B 0,C 180,E1 -3887.552,E2 -3887.552} C_VEL
LIN {X 0,Y 538.014,Z 89.088,A -85,B 0,C 180,E1 -3890.651,E2 -3890.651} C_VEL
LIN {X 0,Y 538.039,Z 89.088,A -85,B 0,C 180,E1 -3893.069,E2 -3893.069} C_VEL
LIN {X 0,Y 538.04,Z 89.089,A -85,B 0,C 180,E1 -3895.681,E2 -3895.681} C_VEL
LIN {X 0,Y 538.025,Z 89.087,A -85,B 0,C 180,E1 -3898.049,E2 -3898.049} C_VEL
LIN {X 0,Y 537.999,Z 89.091,A -85,B 0,C 180,E1 -3900.627,E2 -3900.627} C_VEL
LIN {X 0,Y 538.029,Z 89.092,A -85,B 0,C 180,E1 -3903.288,E2 -3903.288} C_VEL
LIN {X 0,Y 538.008,Z 89.088,A -85,B 0,C 180,E1 -3906.002,E2 -3906.002} C_VEL
LIN {X 0,Y 538.003,Z 89.096,A -85,B 0,C 180,E1 -3908.83,E2 -3908.83} C_VEL
LIN {X 0,Y 538.05,Z 89.091,A -85,B 0,C 180,E1 -3910.774,E2 -3910.774} C_VEL
LIN {X 0,Y 538.002,Z 89.089,A -85,B 0,C 180,E1 -3913.814,E2 -3913.814} C_VEL
LIN {X 0,Y 538.007,Z 89.09,A -85,B 0,C 180,E1 -3916.19,E2 -3916.19} C_VEL
LIN {X 0,Y 538.05,Z 89.084,A -85,B 0,C 180,E1 -3919.251,E2 -3919.251} C_VEL
LIN {X 0,Y 537.976,Z 89.096,A -85,B 0,C 180,E1 -3922.126,E2 -3922.126} C_VEL
LIN {X 0,Y 538,Z 89.092,A -85,B 0,C 180,E1 -3924.92,E2 -3924.92} C_VEL
LIN {X 0,Y 538.009,Z 89.089,A -85,B 0,C 180,E1 -3927.621,E2 -3927.621} C_VEL
LIN {X 0,Y 538.02,Z 89.096,A -85,B 0,C 180,E1 -3930.243,E2 -3930.243} C_VEL
LIN {X 0,Y 538.05,Z 89.085,A -85,B 0,C 180,E1 -3932.799,E2 -3932.799} C_VEL
LIN {X 0,Y 538.04,Z 89.085,A -85,B 0,C 180,E1 -3935.296,E2 -3935.296} C_VEL
LIN {X 0,Y 538.027,Z 89.095,A -85,B 0,C 180,E1 -3938.036,E2 -3938.036} C_VEL
LIN {X 0,Y 538.023,Z 89.086,A -85,B 0,C 180,E1 -3940.943,E2 -3940.943} C_VEL
LIN {X 0,Y 538.013,Z 89.089,A -85,B 0,C 180,E1 -3943.302,E2 -3943.302} C_VEL
LIN {X 0,Y 538.048,Z 89.09,A -85,B 0,C 180,E1 -3945.633,E2 -3945.633} C_VEL
LIN {X 0,Y 538.075,Z 89.08,A -85,B 0,C 180,E1 -3948.704,E2 -3948.704} C_VEL
LIN {X 0,Y 538.08,Z 89.086,A -85,B 0,C 180,E1 -3951.742,E2 -3951.742} C_VEL
LIN {X 0,Y 538.176,Z 89.068,A -85,B 0,C 180,E1 -3954.758,E2 -3954.758} C_VEL
LIN {X 0,Y 538.157,Z 89.074,A -85,B 0,C 180,E1 -3957.757,E2 -3957.757} C_VEL
LIN {X 0,Y 538.178,Z 89.069,A -85,B 0,C 180,E1 -3960.751,E2 -3960.751} C_VEL
LIN {X 0,Y 538.134,Z 89.078,A -85,B 0,C 180,E1 -3962.997,E2 -3962.997} C_VEL
LIN {X 0,Y 538.116,Z 89.075,A -85,B 0,C 180,E1 -3966,E2 -3966} C_VEL
LIN {X 0,Y 538.065,Z 89.09,A -85,B 0,C 180,E1 -3969.02,E2 -3969.02} C_VEL
LIN {X 0,Y 538.076,Z 89.08,A -85,B 0,C 180,E1 -3972.065,E2 -3972.065} C_VEL
LIN {X 0,Y 538.039,Z 89.089,A -85,B 0,C 180,E1 -3975.146,E2 -3975.146} C_VEL
LIN {X 0,Y 538.027,Z 89.088,A -85,B 0,C 180,E1 -3978.272,E2 -3978.272} C_VEL
LIN {X 0,Y 538.035,Z 89.093,A -85,B 0,C 180,E1 -3980.653,E2 -3980.653} C_VEL
LIN {X 0,Y 538.02,Z 89.087,A -85,B 0,C 180,E1 -3983.889,E2 -3983.889} C_VEL
LIN {X 0,Y 538.046,Z 89.09,A -85,B 0,C 180,E1 -3986.368,E2 -3986.368} C_VEL
LIN {X 0,Y 538.028,Z 89.088,A -85,B 0,C 180,E1 -3988.936,E2 -3988.936} C_VEL
LIN {X 0,Y 538.011,Z 89.091,A -85,B 0,C 180,E1 -3991.89,E2 -3991.89} C_VEL
LIN {X 0,Y 538.023,Z 89.09,A -85,B 0,C 180,E1 -3994.622,E2 -3994.622} C_VEL
LIN {X 0,Y 538.004,Z 89.089,A -85,B 0,C 180,E1 -3997.172,E2 -3997.172} C_VEL
LIN {X 0,Y 538.021,Z 89.091,A -85,B 0,C 180,E1 -3999.799,E2 -3999.799} C_VEL
LIN {X 0,Y 538.017,Z 89.088,A -85,B 0,C 180,E1 -4002.788,E2 -4002.788} C_VEL
LIN {X 0,Y 538.03,Z 89.086,A -85,B 0,C 180,E1 -4005.142,E2 -4005.142} C_VEL
LIN {X 0,Y 538.034,Z 89.089,A -85,B 0,C 180,E1 -4008.229,E2 -4008.229} C_VEL
LIN {X 0,Y 538.012,Z 89.089,A -85,B 0,C 180,E1 -4011.171,E2 -4011.171} C_VEL
LIN {X 0,Y 537.993,Z 89.093,A -85,B 0,C 180,E1 -4014.09,E2 -4014.09} C_VEL
LIN {X 0,Y 538.03,Z 89.086,A -85,B 0,C 180,E1 -4016.729,E2 -4016.729} C_VEL
LIN {X 0,Y 538.014,Z 89.097,A -85,B 0,C 180,E1 -4019.56,E2 -4019.56} C_VEL
LIN {X 0,Y 538.04,Z 89.09,A -85,B 0,C 180,E1 -4021.952,E2 -4021.952} C_VEL
LIN {X 0,Y 538.055,Z 89.121,A -85,B 0,C 180,E1 -4024.494,E2 -4024.494} C_VEL
LIN {X 0,Y 539.758,Z 98.029,A -85,B 0,C 180,E1 -4025.858,E2 -4025.858} C_VEL
LIN {X 0,Y 539.332,Z 117.454,A -85,B 0,C 180,E1 -4028.602,E2 -4028.602} C_VEL
LIN {X 0,Y 538.911,Z 138.788,A -85,B 0,C 180,E1 -4031.565,E2 -4031.565} C_VEL
LIN {X 0,Y 538.797,Z 142.803,A -85,B 0,C 180,E1 -4032.116,E2 -4032.116} C_VEL
LIN {X 0,Y 540.666,Z 153.51,A -85,B 0,C 180,E1 -4032.33,E2 -4032.33} C_VEL
LIN {X 0,Y 540.08,Z 281.097,A -85,B 0,C 180,E1 -4034.07,E2 -4034.07} C_VEL
LIN {X 0,Y 539.874,Z 295.588,A -85,B 0,C 180,E1 -4034.424,E2 -4034.424} C_VEL
LIN {X 0,Y 539.626,Z 309.032,A -85,B 0,C 180,E1 -4034.903,E2 -4034.903} C_VEL
LIN {X 0,Y 539.341,Z 321.245,A -85,B 0,C 180,E1 -4035.474,E2 -4035.474} C_VEL
LIN {X 0,Y 539.009,Z 334.096,A -85,B 0,C 180,E1 -4036.235,E2 -4036.235} C_VEL
LIN {X 0,Y 538.694,Z 345.782,A -85,B 0,C 180,E1 -4037.091,E2 -4037.091} C_VEL
LIN {X 0,Y 538.453,Z 356.937,A -85,B 0,C 180,E1 -4038.086,E2 -4038.086} C_VEL
LIN {X 0,Y 538.199,Z 366.288,A -85,B 0,C 180,E1 -4039.087,E2 -4039.087} C_VEL
LIN {X 0,Y 537.958,Z 375.188,A -85,B 0,C 180,E1 -4040.223,E2 -4040.223} C_VEL
LIN {X 0,Y 537.796,Z 383.717,A -85,B 0,C 180,E1 -4041.547,E2 -4041.547} C_VEL
LIN {X 0,Y 537.659,Z 390.591,A -85,B 0,C 180,E1 -4042.868,E2 -4042.868} C_VEL
LIN {X 0,Y 537.635,Z 396.732,A -85,B 0,C 180,E1 -4044.375,E2 -4044.375} C_VEL
LIN {X 0,Y 537.548,Z 400.238,A -85,B 0,C 180,E1 -4045.502,E2 -4045.502} C_VEL
LIN {X 0,Y 537.547,Z 403.65,A -85,B 0,C 180,E1 -4047.003,E2 -4047.003} C_VEL
LIN {X 0,Y 537.448,Z 405.666,A -85,B 0,C 180,E1 -4048.502,E2 -4048.502} C_VEL
LIN {X 0,Y 537.442,Z 406.334,A -85,B 0,C 180,E1 -4050.001,E2 -4050.001} C_VEL
LIN {X 0,Y 537.448,Z 405.664,A -85,B 0,C 180,E1 -4051.5,E2 -4051.5} C_VEL
LIN {X 0,Y 537.547,Z 403.648,A -85,B 0,C 180,E1 -4052.999,E2 -4052.999} C_VEL
LIN {X 0,Y 537.548,Z 400.231,A -85,B 0,C 180,E1 -4054.5,E2 -4054.5} C_VEL
LIN {X 0,Y 537.633,Z 395.315,A -85,B 0,C 180,E1 -4056.004,E2 -4056.004} C_VEL
LIN {X 0,Y 537.662,Z 390.572,A -85,B 0,C 180,E1 -4057.134,E2 -4057.134} C_VEL
LIN {X 0,Y 537.798,Z 383.695,A -85,B 0,C 180,E1 -4058.455,E2 -4058.455} C_VEL
LIN {X 0,Y 537.958,Z 375.158,A -85,B 0,C 180,E1 -4059.779,E2 -4059.779} C_VEL
LIN {X 0,Y 538.213,Z 366.253,A -85,B 0,C 180,E1 -4060.915,E2 -4060.915} C_VEL
LIN {X 0,Y 538.445,Z 355.464,A -85,B 0,C 180,E1 -4062.055,E2 -4062.055} C_VEL
LIN {X 0,Y 538.7,Z 344.549,A -85,B 0,C 180,E1 -4063.007,E2 -4063.007} C_VEL
LIN {X 0,Y 539.011,Z 332.603,A -85,B 0,C 180,E1 -4063.863,E2 -4063.863} C_VEL
LIN {X 0,Y 539.398,Z 319.382,A -85,B 0,C 180,E1 -4064.623,E2 -4064.623} C_VEL
LIN {X 0,Y 539.695,Z 307.232,A -85,B 0,C 180,E1 -4065.17,E2 -4065.17} C_VEL
LIN {X 0,Y 539.873,Z 293.638,A -85,B 0,C 180,E1 -4065.635,E2 -4065.635} C_VEL
LIN {X 0,Y 540.061,Z 279.602,A -85,B 0,C 180,E1 -4065.957,E2 -4065.957} C_VEL
LIN {X 0,Y 540.608,Z 153.121,A -85,B 0,C 180,E1 -4067.677,E2 -4067.677} C_VEL
LIN {X 0,Y 538.809,Z 142.721,A -85,B 0,C 180,E1 -4067.886,E2 -4067.886} C_VEL
LIN {X 0,Y 539.208,Z 121.604,A -85,B 0,C 180,E1 -4070.805,E2 -4070.805} C_VEL
LIN {X 0,Y 539.734,Z 100.266,A -85,B 0,C 180,E1 -4073.808,E2 -4073.808} C_VEL
LIN {X 0,Y 539.556,Z 96.267,A -85,B 0,C 180,E1 -4074.39,E2 -4074.39} C_VEL
LIN {X 0,Y 538.039,Z 89.091,A -85,B 0,C 180,E1 -4075.535,E2 -4075.535} C_VEL
LIN {X 0,Y 538.046,Z 89.088,A -85,B 0,C 180,E1 -4078.051,E2 -4078.051} C_VEL
LIN {X 0,Y 538.022,Z 89.095,A -85,B 0,C 180,E1 -4080.628,E2 -4080.628} C_VEL
LIN {X 0,Y 538.03,Z 89.089,A -85,B 0,C 180,E1 -4083.279,E2 -4083.279} C_VEL
LIN {X 0,Y 538,Z 89.097,A -85,B 0,C 180,E1 -4086.005,E2 -4086.005} C_VEL
LIN {X 0,Y 538.023,Z 89.089,A -85,B 0,C 180,E1 -4088.831,E2 -4088.831} C_VEL
LIN {X 0,Y 538.035,Z 89.09,A -85,B 0,C 180,E1 -4091.774,E2 -4091.774} C_VEL
LIN {X 0,Y 538.009,Z 89.089,A -85,B 0,C 180,E1 -4094.863,E2 -4094.863} C_VEL
LIN {X 0,Y 538.031,Z 89.088,A -85,B 0,C 180,E1 -4097.214,E2 -4097.214} C_VEL
LIN {X 0,Y 538.021,Z 89.089,A -85,B 0,C 180,E1 -4100.201,E2 -4100.201} C_VEL
LIN {X 0,Y 538.031,Z 89.087,A -85,B 0,C 180,E1 -4103.066,E2 -4103.066} C_VEL
LIN {X 0,Y 538.022,Z 89.091,A -85,B 0,C 180,E1 -4105.825,E2 -4105.825} C_VEL
LIN {X 0,Y 538.02,Z 89.087,A -85,B 0,C 180,E1 -4108.498,E2 -4108.498} C_VEL
LIN {X 0,Y 538.031,Z 89.093,A -85,B 0,C 180,E1 -4111.097,E2 -4111.097} C_VEL
LIN {X 0,Y 538.034,Z 89.088,A -85,B 0,C 180,E1 -4113.631,E2 -4113.631} C_VEL
LIN {X 0,Y 538.02,Z 89.085,A -85,B 0,C 180,E1 -4116.121,E2 -4116.121} C_VEL
LIN {X 0,Y 538.049,Z 89.085,A -85,B 0,C 180,E1 -4119.347,E2 -4119.347} C_VEL
LIN {X 0,Y 538.048,Z 89.088,A -85,B 0,C 180,E1 -4122.466,E2 -4122.466} C_VEL
LIN {X 0,Y 538.063,Z 89.082,A -85,B 0,C 180,E1 -4125.629,E2 -4125.629} C_VEL
LIN {X 0,Y 538.087,Z 89.086,A -85,B 0,C 180,E1 -4128.7,E2 -4128.7} C_VEL
LIN {X 0,Y 538.068,Z 89.081,A -85,B 0,C 180,E1 -4131.737,E2 -4131.737} C_VEL
LIN {X 0,Y 538.157,Z 89.074,A -85,B 0,C 180,E1 -4134.753,E2 -4134.753} C_VEL
LIN {X 0,Y 538.172,Z 89.069,A -85,B 0,C 180,E1 -4137.752,E2 -4137.752} C_VEL
LIN {X 0,Y 538.183,Z 89.066,A -85,B 0,C 180,E1 -4140.746,E2 -4140.746} C_VEL
LIN {X 0,Y 538.136,Z 89.073,A -85,B 0,C 180,E1 -4142.992,E2 -4142.992} C_VEL
LIN {X 0,Y 538.117,Z 89.082,A -85,B 0,C 180,E1 -4145.995,E2 -4145.995} C_VEL
LIN {X 0,Y 538.056,Z 89.082,A -85,B 0,C 180,E1 -4149.015,E2 -4149.015} C_VEL
LIN {X 0,Y 538.065,Z 89.084,A -85,B 0,C 180,E1 -4152.06,E2 -4152.06} C_VEL
LIN {X 0,Y 538.041,Z 89.088,A -85,B 0,C 180,E1 -4155.141,E2 -4155.141} C_VEL
LIN {X 0,Y 538.011,Z 89.089,A -85,B 0,C 180,E1 -4158.268,E2 -4158.268} C_VEL
LIN {X 0,Y 538.033,Z 89.085,A -85,B 0,C 180,E1 -4160.648,E2 -4160.648} C_VEL
LIN {X 0,Y 538.001,Z 89.091,A -85,B 0,C 180,E1 -4163.874,E2 -4163.874} C_VEL
LIN {X 0,Y 538.028,Z 89.086,A -85,B 0,C 180,E1 -4166.364,E2 -4166.364} C_VEL
LIN {X 0,Y 538.021,Z 89.093,A -85,B 0,C 180,E1 -4168.93,E2 -4168.93} C_VEL
LIN {X 0,Y 537.998,Z 89.091,A -85,B 0,C 180,E1 -4171.884,E2 -4171.884} C_VEL
LIN {X 0,Y 537.996,Z 89.093,A -85,B 0,C 180,E1 -4174.614,E2 -4174.614} C_VEL
LIN {X 0,Y 537.988,Z 89.092,A -85,B 0,C 180,E1 -4177.166,E2 -4177.166} C_VEL
LIN {X 0,Y 537.992,Z 89.092,A -85,B 0,C 180,E1 -4180.233,E2 -4180.233} C_VEL
LIN {X 0,Y 537.348,Z 89.176,A -85,B 0,C 180,E1 -4180.858,E2 -4180.858} C_VEL
LIN {X 0,Y 534.5,Z 89.529,A -85,B 0,C 180,E1 -4181.873,E2 -4181.873} C_VEL
LIN {X 0,Y 532.074,Z 89.836,A -85,B 0,C 180,E1 -4182.69,E2 -4182.69} C_VEL
LIN {X 0,Y 531.023,Z 89.962,A -85,B 0,C 180,E1 -4183.321,E2 -4183.321} C_VEL
LIN {X 0,Y 530.933,Z 89.972,A -85,B 0,C 180,E1 -4183.535,E2 -4183.535} C_VEL
LIN {X 0,Y 530.923,Z 89.98,A -85,B 0,C 180,E1 -4186.5,E2 -4186.5} C_VEL
LIN {X 0,Y 530.939,Z 89.977,A -85,B 0,C 180,E1 -4188.976,E2 -4188.976} C_VEL
LIN {X 0,Y 530.986,Z 90.161,A -85,B 0,C 180,E1 -4191.564,E2 -4191.564} C_VEL
LIN {X 0,Y 532.249,Z 97.269,A -85,B 0,C 180,E1 -4192.835,E2 -4192.835} C_VEL
LIN {X 0,Y 531.921,Z 112.503,A -85,B 0,C 180,E1 -4195.379,E2 -4195.379} C_VEL
LIN {X 0,Y 531.855,Z 115.995,A -85,B 0,C 180,E1 -4195.941,E2 -4195.941} C_VEL
LIN {X 0,Y 533.951,Z 126.323,A -85,B 0,C 180,E1 -4196.159,E2 -4196.159} C_VEL
LIN {X 0,Y 533.305,Z 252.607,A -85,B 0,C 180,E1 -4197.907,E2 -4197.907} C_VEL
LIN {X 0,Y 533.073,Z 266.759,A -85,B 0,C 180,E1 -4198.255,E2 -4198.255} C_VEL
LIN {X 0,Y 532.83,Z 280.824,A -85,B 0,C 180,E1 -4198.765,E2 -4198.765} C_VEL
LIN {X 0,Y 532.53,Z 293.074,A -85,B 0,C 180,E1 -4199.352,E2 -4199.352} C_VEL
LIN {X 0,Y 532.176,Z 305.392,A -85,B 0,C 180,E1 -4200.096,E2 -4200.096} C_VEL
LIN {X 0,Y 531.818,Z 318.076,A -85,B 0,C 180,E1 -4201.052,E2 -4201.052} C_VEL
LIN {X 0,Y 531.485,Z 329.59,A -85,B 0,C 180,E1 -4202.12,E2 -4202.12} C_VEL
LIN {X 0,Y 531.155,Z 339.688,A -85,B 0,C 180,E1 -4203.264,E2 -4203.264} C_VEL
LIN {X 0,Y 530.931,Z 348.769,A -85,B 0,C 180,E1 -4204.518,E2 -4204.518} C_VEL
LIN {X 0,Y 530.745,Z 356.184,A -85,B 0,C 180,E1 -4205.763,E2 -4205.763} C_VEL
LIN {X 0,Y 530.613,Z 362.223,A -85,B 0,C 180,E1 -4206.999,E2 -4206.999} C_VEL
LIN {X 0,Y 530.532,Z 367.064,A -85,B 0,C 180,E1 -4208.227,E2 -4208.227} C_VEL
LIN {X 0,Y 530.502,Z 370.818,A -85,B 0,C 180,E1 -4209.446,E2 -4209.446} C_VEL
LIN {X 0,Y 530.417,Z 373.627,A -85,B 0,C 180,E1 -4210.654,E2 -4210.654} C_VEL
LIN {X 0,Y 530.356,Z 375.998,A -85,B 0,C 180,E1 -4212.254,E2 -4212.254} C_VEL
LIN {X 0,Y 530.343,Z 376.904,A -85,B 0,C 180,E1 -4213.841,E2 -4213.841} C_VEL
LIN {X 0,Y 530.401,Z 376.389,A -85,B 0,C 180,E1 -4215.418,E2 -4215.418} C_VEL
LIN {X 0,Y 530.414,Z 374.473,A -85,B 0,C 180,E1 -4216.981,E2 -4216.981} C_VEL
LIN {X 0,Y 530.466,Z 371.106,A -85,B 0,C 180,E1 -4218.536,E2 -4218.536} C_VEL
LIN {X 0,Y 530.536,Z 366.241,A -85,B 0,C 180,E1 -4220.083,E2 -4220.083} C_VEL
LIN {X 0,Y 530.612,Z 361.559,A -85,B 0,C 180,E1 -4221.238,E2 -4221.238} C_VEL
LIN {X 0,Y 530.79,Z 354.766,A -85,B 0,C 180,E1 -4222.582,E2 -4222.582} C_VEL
LIN {X 0,Y 530.98,Z 346.382,A -85,B 0,C 180,E1 -4223.921,E2 -4223.921} C_VEL
LIN {X 0,Y 531.214,Z 337.67,A -85,B 0,C 180,E1 -4225.066,E2 -4225.066} C_VEL
LIN {X 0,Y 531.542,Z 327.154,A -85,B 0,C 180,E1 -4226.208,E2 -4226.208} C_VEL
LIN {X 0,Y 531.814,Z 316.596,A -85,B 0,C 180,E1 -4227.158,E2 -4227.158} C_VEL
LIN {X 0,Y 532.163,Z 305.085,A -85,B 0,C 180,E1 -4228.012,E2 -4228.012} C_VEL
LIN {X 0,Y 532.564,Z 292.437,A -85,B 0,C 180,E1 -4228.77,E2 -4228.77} C_VEL
LIN {X 0,Y 532.851,Z 279.392,A -85,B 0,C 180,E1 -4229.385,E2 -4229.385} C_VEL
LIN {X 0,Y 533.073,Z 265.272,A -85,B 0,C 180,E1 -4229.881,E2 -4229.881} C_VEL
LIN {X 0,Y 533.247,Z 251.153,A -85,B 0,C 180,E1 -4230.211,E2 -4230.211} C_VEL
LIN {X 0,Y 533.831,Z 125.617,A -85,B 0,C 180,E1 -4231.944,E2 -4231.944} C_VEL
LIN {X 0,Y 531.83,Z 115.656,A -85,B 0,C 180,E1 -4232.176,E2 -4232.176} C_VEL
LIN {X 0,Y 532.276,Z 97.99,A -85,B 0,C 180,E1 -4235.112,E2 -4235.112} C_VEL
LIN {X 0,Y 531.585,Z 92.519,A -85,B 0,C 180,E1 -4236.07,E2 -4236.07} C_VEL
LIN {X 0,Y 531.03,Z 89.965,A -85,B 0,C 180,E1 -4236.541,E2 -4236.541} C_VEL
LIN {X 0,Y 531.01,Z 89.964,A -85,B 0,C 180,E1 -4239.137,E2 -4239.137} C_VEL
LIN {X 0,Y 531.024,Z 89.968,A -85,B 0,C 180,E1 -4241.679,E2 -4241.679} C_VEL
LIN {X 0,Y 531.039,Z 89.957,A -85,B 0,C 180,E1 -4244.976,E2 -4244.976} C_VEL
LIN {X 0,Y 530.991,Z 89.97,A -85,B 0,C 180,E1 -4247.722,E2 -4247.722} C_VEL
LIN {X 0,Y 530.978,Z 89.966,A -85,B 0,C 180,E1 -4250.938,E2 -4250.938} C_VEL
LIN {X 0,Y 530.989,Z 89.964,A -85,B 0,C 180,E1 -4254.051,E2 -4254.051} C_VEL
LIN {X 0,Y 531.001,Z 89.963,A -85,B 0,C 180,E1 -4256.742,E2 -4256.742} C_VEL
LIN {X 0,Y 530.972,Z 89.973,A -85,B 0,C 180,E1 -4259.322,E2 -4259.322} C_VEL
LIN {X 0,Y 530.96,Z 89.966,A -85,B 0,C 180,E1 -4262.107,E2 -4262.107} C_VEL
LIN {X 0,Y 530.97,Z 89.971,A -85,B 0,C 180,E1 -4264.858,E2 -4264.858} C_VEL
LIN {X 0,Y 530.95,Z 89.97,A -85,B 0,C 180,E1 -4267.507,E2 -4267.507} C_VEL
LIN {X 0,Y 531.01,Z 89.963,A -85,B 0,C 180,E1 -4270.429,E2 -4270.429} C_VEL
LIN {X 0,Y 530.968,Z 89.966,A -85,B 0,C 180,E1 -4273.492,E2 -4273.492} C_VEL
LIN {X 0,Y 530.995,Z 89.971,A -85,B 0,C 180,E1 -4276.713,E2 -4276.713} C_VEL
LIN {X 0,Y 531.003,Z 89.961,A -85,B 0,C 180,E1 -4279.574,E2 -4279.574} C_VEL
LIN {X 0,Y 530.952,Z 89.976,A -85,B 0,C 180,E1 -4282.577,E2 -4282.577} C_VEL
LIN {X 0,Y 530.981,Z 89.964,A -85,B 0,C 180,E1 -4285.314,E2 -4285.314} C_VEL
LIN {X 0,Y 530.961,Z 89.971,A -85,B 0,C 180,E1 -4288.036,E2 -4288.036} C_VEL
LIN {X 0,Y 530.982,Z 89.965,A -85,B 0,C 180,E1 -4290.873,E2 -4290.873} C_VEL
LIN {X 0,Y 530.993,Z 89.962,A -85,B 0,C 180,E1 -4293.26,E2 -4293.26} C_VEL
LIN {X 0,Y 531.005,Z 89.967,A -85,B 0,C 180,E1 -4295.953,E2 -4295.953} C_VEL
LIN {X 0,Y 530.988,Z 89.963,A -85,B 0,C 180,E1 -4299.065,E2 -4299.065} C_VEL
LIN {X 0,Y 530.998,Z 89.965,A -85,B 0,C 180,E1 -4302.28,E2 -4302.28} C_VEL
LIN {X 0,Y 531.002,Z 89.965,A -85,B 0,C 180,E1 -4305.438,E2 -4305.438} C_VEL
LIN {X 0,Y 531.031,Z 89.958,A -85,B 0,C 180,E1 -4308.553,E2 -4308.553} C_VEL
LIN {X 0,Y 531.049,Z 89.964,A -85,B 0,C 180,E1 -4311.632,E2 -4311.632} C_VEL
LIN {X 0,Y 531.131,Z 89.945,A -85,B 0,C 180,E1 -4314.688,E2 -4314.688} C_VEL
LIN {X 0,Y 531.129,Z 89.95,A -85,B 0,C 180,E1 -4317.728,E2 -4317.728} C_VEL
LIN {X 0,Y 531.148,Z 89.945,A -85,B 0,C 180,E1 -4320.761,E2 -4320.761} C_VEL
LIN {X 0,Y 531.101,Z 89.954,A -85,B 0,C 180,E1 -4323.037,E2 -4323.037} C_VEL
LIN {X 0,Y 531.076,Z 89.952,A -85,B 0,C 180,E1 -4326.079,E2 -4326.079} C_VEL
LIN {X 0,Y 531.025,Z 89.966,A -85,B 0,C 180,E1 -4329.14,E2 -4329.14} C_VEL
LIN {X 0,Y 531.034,Z 89.958,A -85,B 0,C 180,E1 -4332.227,E2 -4332.227} C_VEL
LIN {X 0,Y 530.99,Z 89.965,A -85,B 0,C 180,E1 -4335.352,E2 -4335.352} C_VEL
LIN {X 0,Y 530.986,Z 89.968,A -85,B 0,C 180,E1 -4338.523,E2 -4338.523} C_VEL
LIN {X 0,Y 530.995,Z 89.967,A -85,B 0,C 180,E1 -4340.94,E2 -4340.94} C_VEL
LIN {X 0,Y 530.976,Z 89.968,A -85,B 0,C 180,E1 -4344.226,E2 -4344.226} C_VEL
LIN {X 0,Y 531.008,Z 89.966,A -85,B 0,C 180,E1 -4346.745,E2 -4346.745} C_VEL
LIN {X 0,Y 530.978,Z 89.964,A -85,B 0,C 180,E1 -4349.325,E2 -4349.325} C_VEL
LIN {X 0,Y 530.967,Z 89.971,A -85,B 0,C 180,E1 -4352.103,E2 -4352.103} C_VEL
LIN {X 0,Y 530.98,Z 89.965,A -85,B 0,C 180,E1 -4354.855,E2 -4354.855} C_VEL
LIN {X 0,Y 530.964,Z 89.967,A -85,B 0,C 180,E1 -4357.509,E2 -4357.509} C_VEL
LIN {X 0,Y 530.979,Z 89.968,A -85,B 0,C 180,E1 -4360.435,E2 -4360.435} C_VEL
LIN {X 0,Y 530.963,Z 89.968,A -85,B 0,C 180,E1 -4363.496,E2 -4363.496} C_VEL
LIN {X 0,Y 530.954,Z 89.969,A -85,B 0,C 180,E1 -4366.506,E2 -4366.506} C_VEL
LIN {X 0,Y 530.984,Z 89.963,A -85,B 0,C 180,E1 -4368.978,E2 -4368.978} C_VEL
LIN {X 0,Y 530.956,Z 89.972,A -85,B 0,C 180,E1 -4371.531,E2 -4371.531} C_VEL
LIN {X 0,Y 530.953,Z 89.968,A -85,B 0,C 180,E1 -4374.381,E2 -4374.381} C_VEL
LIN {X 0,Y 530.966,Z 89.968,A -85,B 0,C 180,E1 -4377.135,E2 -4377.135} C_VEL
LIN {X 0,Y 530.961,Z 89.973,A -85,B 0,C 180,E1 -4379.804,E2 -4379.804} C_VEL
LIN {X 0,Y 531.013,Z 89.963,A -85,B 0,C 180,E1 -4382.469,E2 -4382.469} C_VEL
LIN {X 0,Y 531.006,Z 90.018,A -85,B 0,C 180,E1 -4384.291,E2 -4384.291} C_VEL
LIN {X 0,Y 532.825,Z 98.971,A -85,B 0,C 180,E1 -4385.688,E2 -4385.688} C_VEL
LIN {X 0,Y 532.455,Z 115.858,A -85,B 0,C 180,E1 -4388.108,E2 -4388.108} C_VEL
LIN {X 0,Y 532.007,Z 135.747,A -85,B 0,C 180,E1 -4390.917,E2 -4390.917} C_VEL
LIN {X 0,Y 531.826,Z 142.595,A -85,B 0,C 180,E1 -4391.872,E2 -4391.872} C_VEL
LIN {X 0,Y 533.873,Z 155.085,A -85,B 0,C 180,E1 -4392.122,E2 -4392.122} C_VEL
LIN {X 0,Y 533.241,Z 280.851,A -85,B 0,C 180,E1 -4393.86,E2 -4393.86} C_VEL
LIN {X 0,Y 533.017,Z 295.171,A -85,B 0,C 180,E1 -4394.213,E2 -4394.213} C_VEL
LIN {X 0,Y 532.764,Z 308.812,A -85,B 0,C 180,E1 -4394.704,E2 -4394.704} C_VEL
LIN {X 0,Y 532.448,Z 321.031,A -85,B 0,C 180,E1 -4395.282,E2 -4395.282} C_VEL
LIN {X 0,Y 532.061,Z 333.885,A -85,B 0,C 180,E1 -4396.052,E2 -4396.052} C_VEL
LIN {X 0,Y 531.692,Z 345.574,A -85,B 0,C 180,E1 -4396.918,E2 -4396.918} C_VEL
LIN {X 0,Y 531.448,Z 356.704,A -85,B 0,C 180,E1 -4397.924,E2 -4397.924} C_VEL
LIN {X 0,Y 531.184,Z 366.086,A -85,B 0,C 180,E1 -4398.941,E2 -4398.941} C_VEL
LIN {X 0,Y 530.903,Z 374.987,A -85,B 0,C 180,E1 -4400.092,E2 -4400.092} C_VEL
LIN {X 0,Y 530.759,Z 382.396,A -85,B 0,C 180,E1 -4401.242,E2 -4401.242} C_VEL
LIN {X 0,Y 530.63,Z 388.573,A -85,B 0,C 180,E1 -4402.39,E2 -4402.39} C_VEL
LIN {X 0,Y 530.551,Z 393.392,A -85,B 0,C 180,E1 -4403.465,E2 -4403.465} C_VEL
LIN {X 0,Y 530.511,Z 397.784,A -85,B 0,C 180,E1 -4404.68,E2 -4404.68} C_VEL
LIN {X 0,Y 530.497,Z 401.929,A -85,B 0,C 180,E1 -4406.203,E2 -4406.203} C_VEL
LIN {X 0,Y 530.41,Z 404.634,A -85,B 0,C 180,E1 -4407.723,E2 -4407.723} C_VEL
LIN {X 0,Y 530.341,Z 405.972,A -85,B 0,C 180,E1 -4409.242,E2 -4409.242} C_VEL
LIN {X 0,Y 530.341,Z 405.971,A -85,B 0,C 180,E1 -4410.76,E2 -4410.76} C_VEL
LIN {X 0,Y 530.411,Z 404.63,A -85,B 0,C 180,E1 -4412.279,E2 -4412.279} C_VEL
LIN {X 0,Y 530.498,Z 401.923,A -85,B 0,C 180,E1 -4413.799,E2 -4413.799} C_VEL
LIN {X 0,Y 530.512,Z 397.768,A -85,B 0,C 180,E1 -4415.322,E2 -4415.322} C_VEL
LIN {X 0,Y 530.576,Z 392.047,A -85,B 0,C 180,E1 -4416.848,E2 -4416.848} C_VEL
LIN {X 0,Y 530.697,Z 385.599,A -85,B 0,C 180,E1 -4418.186,E2 -4418.186} C_VEL
LIN {X 0,Y 530.874,Z 377.587,A -85,B 0,C 180,E1 -4419.526,E2 -4419.526} C_VEL
LIN {X 0,Y 531.081,Z 369.208,A -85,B 0,C 180,E1 -4420.678,E2 -4420.678} C_VEL
LIN {X 0,Y 531.37,Z 359.093,A -85,B 0,C 180,E1 -4421.834,E2 -4421.834} C_VEL
LIN {X 0,Y 531.647,Z 347.866,A -85,B 0,C 180,E1 -4422.891,E2 -4422.891} C_VEL
LIN {X 0,Y 531.992,Z 335.243,A -85,B 0,C 180,E1 -4423.855,E2 -4423.855} C_VEL
LIN {X 0,Y 532.372,Z 322.712,A -85,B 0,C 180,E1 -4424.625,E2 -4424.625} C_VEL
LIN {X 0,Y 532.723,Z 309.826,A -85,B 0,C 180,E1 -4425.251,E2 -4425.251} C_VEL
LIN {X 0,Y 532.978,Z 295.697,A -85,B 0,C 180,E1 -4425.769,E2 -4425.769} C_VEL
LIN {X 0,Y 533.204,Z 281.815,A -85,B 0,C 180,E1 -4426.119,E2 -4426.119} C_VEL
LIN {X 0,Y 533.418,Z 246.432,A -85,B 0,C 180,E1 -4426.629,E2 -4426.629} C_VEL
LIN {X 0,Y 533.814,Z 154.006,A -85,B 0,C 180,E1 -4427.894,E2 -4427.894} C_VEL
LIN {X 0,Y 531.826,Z 142.526,A -85,B 0,C 180,E1 -4428.127,E2 -4428.127} C_VEL
LIN {X 0,Y 532.338,Z 120,A -85,B 0,C 180,E1 -4431.289,E2 -4431.289} C_VEL
LIN {X 0,Y 532.861,Z 101.535,A -85,B 0,C 180,E1 -4433.928,E2 -4433.928} C_VEL
LIN {X 0,Y 532.439,Z 96.679,A -85,B 0,C 180,E1 -4434.655,E2 -4434.655} C_VEL
LIN {X 0,Y 530.996,Z 89.968,A -85,B 0,C 180,E1 -4435.755,E2 -4435.755} C_VEL
LIN {X 0,Y 530.997,Z 89.97,A -85,B 0,C 180,E1 -4438.457,E2 -4438.457} C_VEL
LIN {X 0,Y 530.964,Z 89.971,A -85,B 0,C 180,E1 -4441.08,E2 -4441.08} C_VEL
LIN {X 0,Y 530.968,Z 89.971,A -85,B 0,C 180,E1 -4443.775,E2 -4443.775} C_VEL
LIN {X 0,Y 530.961,Z 89.97,A -85,B 0,C 180,E1 -4446.559,E2 -4446.559} C_VEL
LIN {X 0,Y 530.983,Z 89.966,A -85,B 0,C 180,E1 -4449.445,E2 -4449.445} C_VEL
LIN {X 0,Y 530.981,Z 89.971,A -85,B 0,C 180,E1 -4452.164,E2 -4452.164} C_VEL
LIN {X 0,Y 530.983,Z 89.968,A -85,B 0,C 180,E1 -4455.451,E2 -4455.451} C_VEL
LIN {X 0,Y 531.005,Z 89.956,A -85,B 0,C 180,E1 -4458.564,E2 -4458.564} C_VEL
LIN {X 0,Y 530.966,Z 89.974,A -85,B 0,C 180,E1 -4461.528,E2 -4461.528} C_VEL
LIN {X 0,Y 530.962,Z 89.967,A -85,B 0,C 180,E1 -4464.379,E2 -4464.379} C_VEL
LIN {X 0,Y 530.979,Z 89.969,A -85,B 0,C 180,E1 -4467.133,E2 -4467.133} C_VEL
LIN {X 0,Y 530.966,Z 89.969,A -85,B 0,C 180,E1 -4469.801,E2 -4469.801} C_VEL
LIN {X 0,Y 530.98,Z 89.963,A -85,B 0,C 180,E1 -4472.476,E2 -4472.476} C_VEL
LIN {X 0,Y 530.999,Z 89.969,A -85,B 0,C 180,E1 -4474.94,E2 -4474.94} C_VEL
LIN {X 0,Y 530.984,Z 89.965,A -85,B 0,C 180,E1 -4478.245,E2 -4478.245} C_VEL
LIN {X 0,Y 530.995,Z 89.965,A -85,B 0,C 180,E1 -4480.675,E2 -4480.675} C_VEL
LIN {X 0,Y 530.975,Z 89.968,A -85,B 0,C 180,E1 -4483.069,E2 -4483.069} C_VEL
LIN {X 0,Y 531.02,Z 89.96,A -85,B 0,C 180,E1 -4485.434,E2 -4485.434} C_VEL
LIN {X 0,Y 531.045,Z 89.961,A -85,B 0,C 180,E1 -4488.548,E2 -4488.548} C_VEL
LIN {X 0,Y 531.043,Z 89.956,A -85,B 0,C 180,E1 -4491.627,E2 -4491.627} C_VEL
LIN {X 0,Y 531.115,Z 89.952,A -85,B 0,C 180,E1 -4494.683,E2 -4494.683} C_VEL
LIN {X 0,Y 531.144,Z 89.944,A -85,B 0,C 180,E1 -4497.723,E2 -4497.723} C_VEL
LIN {X 0,Y 531.154,Z 89.941,A -85,B 0,C 180,E1 -4500.756,E2 -4500.756} C_VEL
LIN {X 0,Y 531.104,Z 89.949,A -85,B 0,C 180,E1 -4503.032,E2 -4503.032} C_VEL
LIN {X 0,Y 531.072,Z 89.959,A -85,B 0,C 180,E1 -4506.075,E2 -4506.075} C_VEL
LIN {X 0,Y 531.018,Z 89.959,A -85,B 0,C 180,E1 -4509.136,E2 -4509.136} C_VEL
LIN {X 0,Y 531.051,Z 89.964,A -85,B 0,C 180,E1 -4511.667,E2 -4511.667} C_VEL
LIN {X 0,Y 531.029,Z 89.96,A -85,B 0,C 180,E1 -4514.951,E2 -4514.951} C_VEL
LIN {X 0,Y 530.978,Z 89.97,A -85,B 0,C 180,E1 -4517.72,E2 -4517.72} C_VEL
LIN {X 0,Y 531.021,Z 89.958,A -85,B 0,C 180,E1 -4520.124,E2 -4520.124} C_VEL
LIN {X 0,Y 530.939,Z 89.97,A -85,B 0,C 180,E1 -4522.57,E2 -4522.57} C_VEL
LIN {X 0,Y 530.961,Z 89.974,A -85,B 0,C 180,E1 -4525.056,E2 -4525.056} C_VEL
LIN {X 0,Y 531.002,Z 89.964,A -85,B 0,C 180,E1 -4527.592,E2 -4527.592} C_VEL
LIN {X 0,Y 530.955,Z 89.967,A -85,B 0,C 180,E1 -4530.64,E2 -4530.64} C_VEL
LIN {X 0,Y 530.95,Z 89.967,A -85,B 0,C 180,E1 -4533.496,E2 -4533.496} C_VEL
LIN {X 0,Y 530.931,Z 89.973,A -85,B 0,C 180,E1 -4536.15,E2 -4536.15} C_VEL
LIN {X 0,Y 530.947,Z 89.974,A -85,B 0,C 180,E1 -4538.65,E2 -4538.65} C_VEL
LIN {X 0,Y 530.979,Z 89.965,A -85,B 0,C 180,E1 -4541.432,E2 -4541.432} C_VEL
LIN {X 0,Y 530.933,Z 89.972,A -85,B 0,C 180,E1 -4543.535,E2 -4543.535} C_VEL
LIN {X 0,Y 530.257,Z 90.061,A -85,B 0,C 180,E1 -4544.169,E2 -4544.169} C_VEL
LIN {X 0,Y 527.403,Z 90.417,A -85,B 0,C 180,E1 -4545.197,E2 -4545.197} C_VEL
LIN {X 0,Y 524.996,Z 90.718,A -85,B 0,C 180,E1 -4546.026,E2 -4546.026} C_VEL
LIN {X 0,Y 523.963,Z 90.846,A -85,B 0,C 180,E1 -4546.665,E2 -4546.665} C_VEL
LIN {X 0,Y 523.878,Z 90.853,A -85,B 0,C 180,E1 -4546.882,E2 -4546.882} C_VEL
LIN {X 0,Y 523.91,Z 90.857,A -85,B 0,C 180,E1 -4549.916,E2 -4549.916} C_VEL
LIN {X 0,Y 523.939,Z 90.959,A -85,B 0,C 180,E1 -4551.348,E2 -4551.348} C_VEL
LIN {X 0,Y 525.347,Z 98.648,A -85,B 0,C 180,E1 -4552.745,E2 -4552.745} C_VEL
LIN {X 0,Y 524.927,Z 115.651,A -85,B 0,C 180,E1 -4555.622,E2 -4555.622} C_VEL
LIN {X 0,Y 524.917,Z 116.115,A -85,B 0,C 180,E1 -4555.692,E2 -4555.692} C_VEL
LIN {X 0,Y 527.19,Z 126.876,A -85,B 0,C 180,E1 -4555.927,E2 -4555.927} C_VEL
LIN {X 0,Y 526.512,Z 252.564,A -85,B 0,C 180,E1 -4557.689,E2 -4557.689} C_VEL
LIN {X 0,Y 526.26,Z 267.033,A -85,B 0,C 180,E1 -4558.049,E2 -4558.049} C_VEL
LIN {X 0,Y 526.018,Z 280.456,A -85,B 0,C 180,E1 -4558.539,E2 -4558.539} C_VEL
LIN {X 0,Y 525.644,Z 293.54,A -85,B 0,C 180,E1 -4559.171,E2 -4559.171} C_VEL
LIN {X 0,Y 525.246,Z 306.786,A -85,B 0,C 180,E1 -4559.993,E2 -4559.993} C_VEL
LIN {X 0,Y 524.913,Z 318.108,A -85,B 0,C 180,E1 -4560.865,E2 -4560.865} C_VEL
LIN {X 0,Y 524.532,Z 329.425,A -85,B 0,C 180,E1 -4561.924,E2 -4561.924} C_VEL
LIN {X 0,Y 524.173,Z 339.691,A -85,B 0,C 180,E1 -4563.094,E2 -4563.094} C_VEL
LIN {X 0,Y 523.904,Z 348.241,A -85,B 0,C 180,E1 -4564.275,E2 -4564.275} C_VEL
LIN {X 0,Y 523.695,Z 356.526,A -85,B 0,C 180,E1 -4565.679,E2 -4565.679} C_VEL
LIN {X 0,Y 523.544,Z 363.182,A -85,B 0,C 180,E1 -4567.088,E2 -4567.088} C_VEL
LIN {X 0,Y 523.458,Z 367.87,A -85,B 0,C 180,E1 -4568.332,E2 -4568.332} C_VEL
LIN {X 0,Y 523.413,Z 371.513,A -85,B 0,C 180,E1 -4569.566,E2 -4569.566} C_VEL
LIN {X 0,Y 523.346,Z 373.4,A -85,B 0,C 180,E1 -4570.382,E2 -4570.382} C_VEL
LIN {X 0,Y 523.263,Z 375.963,A -85,B 0,C 180,E1 -4572.005,E2 -4572.005} C_VEL
LIN {X 0,Y 523.245,Z 377.054,A -85,B 0,C 180,E1 -4573.616,E2 -4573.616} C_VEL
LIN {X 0,Y 523.301,Z 376.721,A -85,B 0,C 180,E1 -4575.215,E2 -4575.215} C_VEL
LIN {X 0,Y 523.312,Z 374.993,A -85,B 0,C 180,E1 -4576.802,E2 -4576.802} C_VEL
LIN {X 0,Y 523.385,Z 371.856,A -85,B 0,C 180,E1 -4578.379,E2 -4578.379} C_VEL
LIN {X 0,Y 523.453,Z 367.227,A -85,B 0,C 180,E1 -4579.947,E2 -4579.947} C_VEL
LIN {X 0,Y 523.572,Z 360.946,A -85,B 0,C 180,E1 -4581.508,E2 -4581.508} C_VEL
LIN {X 0,Y 523.772,Z 353.971,A -85,B 0,C 180,E1 -4582.869,E2 -4582.869} C_VEL
LIN {X 0,Y 523.977,Z 345.383,A -85,B 0,C 180,E1 -4584.225,E2 -4584.225} C_VEL
LIN {X 0,Y 524.265,Z 336.43,A -85,B 0,C 180,E1 -4585.386,E2 -4585.386} C_VEL
LIN {X 0,Y 524.651,Z 325.627,A -85,B 0,C 180,E1 -4586.543,E2 -4586.543} C_VEL
LIN {X 0,Y 524.983,Z 314.713,A -85,B 0,C 180,E1 -4587.505,E2 -4587.505} C_VEL
LIN {X 0,Y 525.363,Z 302.734,A -85,B 0,C 180,E1 -4588.37,E2 -4588.37} C_VEL
LIN {X 0,Y 525.778,Z 289.351,A -85,B 0,C 180,E1 -4589.137,E2 -4589.137} C_VEL
LIN {X 0,Y 526.067,Z 276.473,A -85,B 0,C 180,E1 -4589.712,E2 -4589.712} C_VEL
LIN {X 0,Y 526.324,Z 262.615,A -85,B 0,C 180,E1 -4590.166,E2 -4590.166} C_VEL
LIN {X 0,Y 526.458,Z 248.173,A -85,B 0,C 180,E1 -4590.477,E2 -4590.477} C_VEL
LIN {X 0,Y 527.178,Z 127.082,A -85,B 0,C 180,E1 -4592.16,E2 -4592.16} C_VEL
LIN {X 0,Y 524.905,Z 115.851,A -85,B 0,C 180,E1 -4592.421,E2 -4592.421} C_VEL
LIN {X 0,Y 525.405,Z 98.311,A -85,B 0,C 180,E1 -4595.372,E2 -4595.372} C_VEL
LIN {X 0,Y 524.001,Z 90.84,A -85,B 0,C 180,E1 -4596.754,E2 -4596.754} C_VEL
LIN {X 0,Y 523.977,Z 90.841,A -85,B 0,C 180,E1 -4599.261,E2 -4599.261} C_VEL
LIN {X 0,Y 523.984,Z 90.845,A -85,B 0,C 180,E1 -4601.751,E2 -4601.751} C_VEL
LIN {X 0,Y 523.993,Z 90.836,A -85,B 0,C 180,E1 -4605.069,E2 -4605.069} C_VEL
LIN {X 0,Y 523.934,Z 90.845,A -85,B 0,C 180,E1 -4607.969,E2 -4607.969} C_VEL
LIN {X 0,Y 523.938,Z 90.841,A -85,B 0,C 180,E1 -4610.41,E2 -4610.41} C_VEL
LIN {X 0,Y 523.934,Z 90.843,A -85,B 0,C 180,E1 -4612.891,E2 -4612.891} C_VEL
LIN {X 0,Y 523.959,Z 90.847,A -85,B 0,C 180,E1 -4615.417,E2 -4615.417} C_VEL
LIN {X 0,Y 523.938,Z 90.842,A -85,B 0,C 180,E1 -4617.999,E2 -4617.999} C_VEL
LIN {X 0,Y 523.936,Z 90.845,A -85,B 0,C 180,E1 -4620.861,E2 -4620.861} C_VEL
LIN {X 0,Y 523.938,Z 90.842,A -85,B 0,C 180,E1 -4623.739,E2 -4623.739} C_VEL
LIN {X 0,Y 523.919,Z 90.845,A -85,B 0,C 180,E1 -4626.411,E2 -4626.411} C_VEL
LIN {X 0,Y 523.945,Z 90.847,A -85,B 0,C 180,E1 -4629.081,E2 -4629.081} C_VEL
LIN {X 0,Y 523.95,Z 90.842,A -85,B 0,C 180,E1 -4631.316,E2 -4631.316} C_VEL
LIN {X 0,Y 523.925,Z 90.845,A -85,B 0,C 180,E1 -4634.228,E2 -4634.228} C_VEL
LIN {X 0,Y 523.939,Z 90.848,A -85,B 0,C 180,E1 -4636.84,E2 -4636.84} C_VEL
LIN {X 0,Y 523.985,Z 90.836,A -85,B 0,C 180,E1 -4639.929,E2 -4639.929} C_VEL
LIN {X 0,Y 523.894,Z 90.85,A -85,B 0,C 180,E1 -4642.871,E2 -4642.871} C_VEL
LIN {X 0,Y 523.921,Z 90.844,A -85,B 0,C 180,E1 -4645.713,E2 -4645.713} C_VEL
LIN {X 0,Y 523.91,Z 90.852,A -85,B 0,C 180,E1 -4648.459,E2 -4648.459} C_VEL
LIN {X 0,Y 523.927,Z 90.842,A -85,B 0,C 180,E1 -4651.129,E2 -4651.129} C_VEL
LIN {X 0,Y 523.966,Z 90.844,A -85,B 0,C 180,E1 -4653.981,E2 -4653.981} C_VEL
LIN {X 0,Y 523.949,Z 90.846,A -85,B 0,C 180,E1 -4656.275,E2 -4656.275} C_VEL
LIN {X 0,Y 523.939,Z 90.841,A -85,B 0,C 180,E1 -4658.77,E2 -4658.77} C_VEL
LIN {X 0,Y 523.936,Z 90.842,A -85,B 0,C 180,E1 -4661.224,E2 -4661.224} C_VEL
LIN {X 0,Y 523.925,Z 90.848,A -85,B 0,C 180,E1 -4663.642,E2 -4663.642} C_VEL
LIN {X 0,Y 523.926,Z 90.848,A -85,B 0,C 180,E1 -4666.031,E2 -4666.031} C_VEL
LIN {X 0,Y 523.996,Z 90.835,A -85,B 0,C 180,E1 -4668.397,E2 -4668.397} C_VEL
LIN {X 0,Y 523.996,Z 90.841,A -85,B 0,C 180,E1 -4671.519,E2 -4671.519} C_VEL
LIN {X 0,Y 524.089,Z 90.822,A -85,B 0,C 180,E1 -4674.616,E2 -4674.616} C_VEL
LIN {X 0,Y 524.101,Z 90.826,A -85,B 0,C 180,E1 -4677.697,E2 -4677.697} C_VEL
LIN {X 0,Y 524.117,Z 90.82,A -85,B 0,C 180,E1 -4680.771,E2 -4680.771} C_VEL
LIN {X 0,Y 524.067,Z 90.831,A -85,B 0,C 180,E1 -4683.077,E2 -4683.077} C_VEL
LIN {X 0,Y 524.038,Z 90.829,A -85,B 0,C 180,E1 -4686.161,E2 -4686.161} C_VEL
LIN {X 0,Y 523.993,Z 90.84,A -85,B 0,C 180,E1 -4689.264,E2 -4689.264} C_VEL
LIN {X 0,Y 523.996,Z 90.834,A -85,B 0,C 180,E1 -4691.742,E2 -4691.742} C_VEL
LIN {X 0,Y 523.986,Z 90.841,A -85,B 0,C 180,E1 -4695.055,E2 -4695.055} C_VEL
LIN {X 0,Y 523.959,Z 90.839,A -85,B 0,C 180,E1 -4697.971,E2 -4697.971} C_VEL
LIN {X 0,Y 523.967,Z 90.842,A -85,B 0,C 180,E1 -4700.412,E2 -4700.412} C_VEL
LIN {X 0,Y 523.912,Z 90.849,A -85,B 0,C 180,E1 -4702.895,E2 -4702.895} C_VEL
LIN {X 0,Y 523.951,Z 90.84,A -85,B 0,C 180,E1 -4705.421,E2 -4705.421} C_VEL
LIN {X 0,Y 523.968,Z 90.84,A -85,B 0,C 180,E1 -4708.001,E2 -4708.001} C_VEL
LIN {X 0,Y 523.941,Z 90.843,A -85,B 0,C 180,E1 -4710.857,E2 -4710.857} C_VEL
LIN {X 0,Y 523.958,Z 90.84,A -85,B 0,C 180,E1 -4713.737,E2 -4713.737} C_VEL
LIN {X 0,Y 523.917,Z 90.85,A -85,B 0,C 180,E1 -4716.406,E2 -4716.406} C_VEL
LIN {X 0,Y 523.918,Z 90.844,A -85,B 0,C 180,E1 -4719.087,E2 -4719.087} C_VEL
LIN {X 0,Y 523.953,Z 90.847,A -85,B 0,C 180,E1 -4722.12,E2 -4722.12} C_VEL
LIN {X 0,Y 523.953,Z 90.84,A -85,B 0,C 180,E1 -4725.311,E2 -4725.311} C_VEL
LIN {X 0,Y 523.957,Z 90.839,A -85,B 0,C 180,E1 -4728.691,E2 -4728.691} C_VEL
LIN {X 0,Y 523.916,Z 90.845,A -85,B 0,C 180,E1 -4731.082,E2 -4731.082} C_VEL
LIN {X 0,Y 523.9,Z 90.853,A -85,B 0,C 180,E1 -4733.827,E2 -4733.827} C_VEL
LIN {X 0,Y 523.941,Z 90.841,A -85,B 0,C 180,E1 -4736.637,E2 -4736.637} C_VEL
LIN {X 0,Y 523.949,Z 90.847,A -85,B 0,C 180,E1 -4739.357,E2 -4739.357} C_VEL
LIN {X 0,Y 523.977,Z 90.84,A -85,B 0,C 180,E1 -4742.283,E2 -4742.283} C_VEL
LIN {X 0,Y 523.983,Z 90.914,A -85,B 0,C 180,E1 -4744.086,E2 -4744.086} C_VEL
LIN {X 0,Y 525.89,Z 100.003,A -85,B 0,C 180,E1 -4745.527,E2 -4745.527} C_VEL
LIN {X 0,Y 525.68,Z 112.108,A -85,B 0,C 180,E1 -4747.294,E2 -4747.294} C_VEL
LIN {X 0,Y 525.128,Z 132.728,A -85,B 0,C 180,E1 -4750.25,E2 -4750.25} C_VEL
LIN {X 0,Y 524.889,Z 142.356,A -85,B 0,C 180,E1 -4751.617,E2 -4751.617} C_VEL
LIN {X 0,Y 527.112,Z 155.769,A -85,B 0,C 180,E1 -4751.897,E2 -4751.897} C_VEL
LIN {X 0,Y 526.407,Z 280.604,A -85,B 0,C 180,E1 -4753.644,E2 -4753.644} C_VEL
LIN {X 0,Y 526.163,Z 295.276,A -85,B 0,C 180,E1 -4754.013,E2 -4754.013} C_VEL
LIN {X 0,Y 525.887,Z 308.59,A -85,B 0,C 180,E1 -4754.499,E2 -4754.499} C_VEL
LIN {X 0,Y 525.553,Z 320.817,A -85,B 0,C 180,E1 -4755.084,E2 -4755.084} C_VEL
LIN {X 0,Y 525.139,Z 333.675,A -85,B 0,C 180,E1 -4755.864,E2 -4755.864} C_VEL
LIN {X 0,Y 524.709,Z 345.366,A -85,B 0,C 180,E1 -4756.741,E2 -4756.741} C_VEL
LIN {X 0,Y 524.436,Z 356.253,A -85,B 0,C 180,E1 -4757.735,E2 -4757.735} C_VEL
LIN {X 0,Y 524.151,Z 365.883,A -85,B 0,C 180,E1 -4758.79,E2 -4758.79} C_VEL
LIN {X 0,Y 523.849,Z 374.785,A -85,B 0,C 180,E1 -4759.957,E2 -4759.957} C_VEL
LIN {X 0,Y 523.709,Z 382.197,A -85,B 0,C 180,E1 -4761.123,E2 -4761.123} C_VEL
LIN {X 0,Y 523.563,Z 388.375,A -85,B 0,C 180,E1 -4762.287,E2 -4762.287} C_VEL
LIN {X 0,Y 523.469,Z 393.592,A -85,B 0,C 180,E1 -4763.473,E2 -4763.473} C_VEL
LIN {X 0,Y 523.443,Z 397.588,A -85,B 0,C 180,E1 -4764.608,E2 -4764.608} C_VEL
LIN {X 0,Y 523.419,Z 401.734,A -85,B 0,C 180,E1 -4766.152,E2 -4766.152} C_VEL
LIN {X 0,Y 523.334,Z 404.439,A -85,B 0,C 180,E1 -4767.692,E2 -4767.692} C_VEL
LIN {X 0,Y 523.247,Z 405.777,A -85,B 0,C 180,E1 -4769.232,E2 -4769.232} C_VEL
LIN {X 0,Y 523.247,Z 405.775,A -85,B 0,C 180,E1 -4770.771,E2 -4770.771} C_VEL
LIN {X 0,Y 523.334,Z 404.434,A -85,B 0,C 180,E1 -4772.31,E2 -4772.31} C_VEL
LIN {X 0,Y 523.42,Z 401.725,A -85,B 0,C 180,E1 -4773.851,E2 -4773.851} C_VEL
LIN {X 0,Y 523.444,Z 397.569,A -85,B 0,C 180,E1 -4775.394,E2 -4775.394} C_VEL
LIN {X 0,Y 523.498,Z 391.845,A -85,B 0,C 180,E1 -4776.941,E2 -4776.941} C_VEL
LIN {X 0,Y 523.618,Z 385.393,A -85,B 0,C 180,E1 -4778.297,E2 -4778.297} C_VEL
LIN {X 0,Y 523.821,Z 377.379,A -85,B 0,C 180,E1 -4779.656,E2 -4779.656} C_VEL
LIN {X 0,Y 524.074,Z 368.998,A -85,B 0,C 180,E1 -4780.822,E2 -4780.822} C_VEL
LIN {X 0,Y 524.385,Z 358.301,A -85,B 0,C 180,E1 -4782.056,E2 -4782.056} C_VEL
LIN {X 0,Y 524.678,Z 347.649,A -85,B 0,C 180,E1 -4783.065,E2 -4783.065} C_VEL
LIN {X 0,Y 525.009,Z 336.451,A -85,B 0,C 180,E1 -4783.944,E2 -4783.944} C_VEL
LIN {X 0,Y 525.411,Z 324.257,A -85,B 0,C 180,E1 -4784.724,E2 -4784.724} C_VEL
LIN {X 0,Y 525.818,Z 310.724,A -85,B 0,C 180,E1 -4785.406,E2 -4785.406} C_VEL
LIN {X 0,Y 526.122,Z 296.153,A -85,B 0,C 180,E1 -4785.957,E2 -4785.957} C_VEL
LIN {X 0,Y 526.377,Z 281.55,A -85,B 0,C 180,E1 -4786.334,E2 -4786.334} C_VEL
LIN {X 0,Y 526.673,Z 242.564,A -85,B 0,C 180,E1 -4786.898,E2 -4786.898} C_VEL
LIN {X 0,Y 527.059,Z 154.848,A -85,B 0,C 180,E1 -4788.117,E2 -4788.117} C_VEL
LIN {X 0,Y 524.882,Z 142.255,A -85,B 0,C 180,E1 -4788.384,E2 -4788.384} C_VEL
LIN {X 0,Y 525.462,Z 119.832,A -85,B 0,C 180,E1 -4791.582,E2 -4791.582} C_VEL
LIN {X 0,Y 525.968,Z 101.401,A -85,B 0,C 180,E1 -4794.261,E2 -4794.261} C_VEL
LIN {X 0,Y 524.987,Z 95.733,A -85,B 0,C 180,E1 -4795.154,E2 -4795.154} C_VEL
LIN {X 0,Y 523.955,Z 90.847,A -85,B 0,C 180,E1 -4795.976,E2 -4795.976} C_VEL
LIN {X 0,Y 523.945,Z 90.847,A -85,B 0,C 180,E1 -4798.875,E2 -4798.875} C_VEL
LIN {X 0,Y 523.929,Z 90.847,A -85,B 0,C 180,E1 -4801.545,E2 -4801.545} C_VEL
LIN {X 0,Y 523.93,Z 90.85,A -85,B 0,C 180,E1 -4804.291,E2 -4804.291} C_VEL
LIN {X 0,Y 523.916,Z 90.844,A -85,B 0,C 180,E1 -4807.133,E2 -4807.133} C_VEL
LIN {X 0,Y 523.95,Z 90.844,A -85,B 0,C 180,E1 -4810.13,E2 -4810.13} C_VEL
LIN {X 0,Y 523.929,Z 90.845,A -85,B 0,C 180,E1 -4812.457,E2 -4812.457} C_VEL
LIN {X 0,Y 523.952,Z 90.842,A -85,B 0,C 180,E1 -4815.31,E2 -4815.31} C_VEL
LIN {X 0,Y 523.968,Z 90.832,A -85,B 0,C 180,E1 -4818.69,E2 -4818.69} C_VEL
LIN {X 0,Y 523.925,Z 90.847,A -85,B 0,C 180,E1 -4821.897,E2 -4821.897} C_VEL
LIN {X 0,Y 523.934,Z 90.844,A -85,B 0,C 180,E1 -4824.911,E2 -4824.911} C_VEL
LIN {X 0,Y 523.947,Z 90.844,A -85,B 0,C 180,E1 -4827.679,E2 -4827.679} C_VEL
LIN {X 0,Y 523.964,Z 90.84,A -85,B 0,C 180,E1 -4830.676,E2 -4830.676} C_VEL
LIN {X 0,Y 523.944,Z 90.843,A -85,B 0,C 180,E1 -4833.725,E2 -4833.725} C_VEL
LIN {X 0,Y 523.923,Z 90.841,A -85,B 0,C 180,E1 -4836.268,E2 -4836.268} C_VEL
LIN {X 0,Y 523.957,Z 90.845,A -85,B 0,C 180,E1 -4838.765,E2 -4838.765} C_VEL
LIN {X 0,Y 523.95,Z 90.844,A -85,B 0,C 180,E1 -4841.219,E2 -4841.219} C_VEL
LIN {X 0,Y 523.933,Z 90.84,A -85,B 0,C 180,E1 -4843.637,E2 -4843.637} C_VEL
LIN {X 0,Y 523.939,Z 90.843,A -85,B 0,C 180,E1 -4846.026,E2 -4846.026} C_VEL
LIN {X 0,Y 524.024,Z 90.835,A -85,B 0,C 180,E1 -4848.392,E2 -4848.392} C_VEL
LIN {X 0,Y 523.995,Z 90.834,A -85,B 0,C 180,E1 -4851.514,E2 -4851.514} C_VEL
LIN {X 0,Y 524.075,Z 90.83,A -85,B 0,C 180,E1 -4854.611,E2 -4854.611} C_VEL
LIN {X 0,Y 524.117,Z 90.819,A -85,B 0,C 180,E1 -4857.692,E2 -4857.692} C_VEL
LIN {X 0,Y 524.125,Z 90.816,A -85,B 0,C 180,E1 -4860.766,E2 -4860.766} C_VEL
LIN {X 0,Y 524.045,Z 90.828,A -85,B 0,C 180,E1 -4863.072,E2 -4863.072} C_VEL
LIN {X 0,Y 524.03,Z 90.835,A -85,B 0,C 180,E1 -4866.156,E2 -4866.156} C_VEL
LIN {X 0,Y 523.988,Z 90.836,A -85,B 0,C 180,E1 -4869.259,E2 -4869.259} C_VEL
LIN {X 0,Y 524.001,Z 90.841,A -85,B 0,C 180,E1 -4871.734,E2 -4871.734} C_VEL
LIN {X 0,Y 523.991,Z 90.837,A -85,B 0,C 180,E1 -4875.048,E2 -4875.048} C_VEL
LIN {X 0,Y 523.943,Z 90.844,A -85,B 0,C 180,E1 -4877.966,E2 -4877.966} C_VEL
LIN {X 0,Y 523.954,Z 90.838,A -85,B 0,C 180,E1 -4880.407,E2 -4880.407} C_VEL
LIN {X 0,Y 523.904,Z 90.85,A -85,B 0,C 180,E1 -4882.89,E2 -4882.89} C_VEL
LIN {X 0,Y 523.907,Z 90.849,A -85,B 0,C 180,E1 -4885.417,E2 -4885.417} C_VEL
LIN {X 0,Y 523.949,Z 90.84,A -85,B 0,C 180,E1 -4887.996,E2 -4887.996} C_VEL
LIN {X 0,Y 523.928,Z 90.845,A -85,B 0,C 180,E1 -4890.85,E2 -4890.85} C_VEL
LIN {X 0,Y 523.917,Z 90.842,A -85,B 0,C 180,E1 -4893.726,E2 -4893.726} C_VEL
LIN {X 0,Y 523.888,Z 90.853,A -85,B 0,C 180,E1 -4896.398,E2 -4896.398} C_VEL
LIN {X 0,Y 523.896,Z 90.851,A -85,B 0,C 180,E1 -4899.082,E2 -4899.082} C_VEL
LIN {X 0,Y 523.936,Z 90.846,A -85,B 0,C 180,E1 -4902.115,E2 -4902.115} C_VEL
LIN {X 0,Y 523.922,Z 90.844,A -85,B 0,C 180,E1 -4905.307,E2 -4905.307} C_VEL
LIN {X 0,Y 523.878,Z 90.853,A -85,B 0,C 180,E1 -4906.882,E2 -4906.882} C_VEL
LIN {X 0,Y 523.206,Z 90.936,A -85,B 0,C 180,E1 -4907.523,E2 -4907.523} C_VEL
LIN {X 0,Y 520.342,Z 91.299,A -85,B 0,C 180,E1 -4908.565,E2 -4908.565} C_VEL
